gfCNCPoint2[4835] = {X 398.4217, Y 43.2753, Z -2.1667, A 0.000, B 0.000, C 0.000 }
gfCNCPoint2[4836] = {X 398.7237, Y 42.4397, Z -2.1667, A 0.000, B 0.000, C 0.000 }
gfCNCPoint2[4837] = {X 399.2028, Y 41.6913, Z -2.1667, A 0.000, B 0.000, C 0.000 }
gfCNCPoint2[4838] = {X 399.8352, Y 41.0672, Z -2.1667, A 0.000, B 0.000, C 0.000 }
gfCNCPoint2[4839] = {X 399.8352, Y 31.6238, Z -2.1667, A 0.000, B 0.000, C 0.000 }
gfCNCPoint2[4840] = {X 399.8383, Y 31.5919, Z -2.1667, A 0.000, B 0.000, C 0.000 }
gfCNCPoint2[4841] = {X 393.5981, Y 20.7408, Z -2.1667, A 0.000, B 0.000, C 0.000 }
gfCNCPoint2[4842] = {X 392.7769, Y 19.3501, Z -2.1667, A 0.000, B 0.000, C 0.000 }
gfCNCPoint2[4843] = {X 391.9239, Y 17.9787, Z -2.1667, A 0.000, B 0.000, C 0.000 }
gfCNCPoint2[4844] = {X 391.4254, Y 17.2996, Z -2.1667, A 0.000, B 0.000, C 0.000 }
gfCNCPoint2[4845] = {X 390.8426, Y 16.6913, Z -2.1667, A 0.000, B 0.000, C 0.000 }
gfCNCPoint2[4846] = {X 390.0091, Y 16.2361, Z -2.1667, A 0.000, B 0.000, C 0.000 }
gfCNCPoint2[4847] = {X 389.3064, Y 15.5972, Z -2.1667, A 0.000, B 0.000, C 0.000 }
gfCNCPoint2[4848] = {X 388.7742, Y 14.8107, Z -2.1667, A 0.000, B 0.000, C 0.000 }
gfCNCPoint2[4849] = {X 388.4423, Y 13.9209, Z -2.1667, A 0.000, B 0.000, C 0.000 }
gfCNCPoint2[4850] = {X 388.3296, Y 12.9779, Z -2.1667, A 0.000, B 0.000, C 0.000 }
gfCNCPoint2[4851] = {X 388.3296, Y 12.1868, Z -2.1667, A 0.000, B 0.000, C 0.000 }
gfCNCPoint2[4852] = {X 388.4299, Y 11.2967, Z -2.1667, A 0.000, B 0.000, C 0.000 }
gfCNCPoint2[4853] = {X 388.7258, Y 10.4513, Z -2.1667, A 0.000, B 0.000, C 0.000 }
gfCNCPoint2[4854] = {X 389.2023, Y 9.6929, Z -2.1667, A 0.000, B 0.000, C 0.000 }
gfCNCPoint2[4855] = {X 389.8357, Y 9.0595, Z -2.1667, A 0.000, B 0.000, C 0.000 }
gfCNCPoint2[4856] = {X 390.5941, Y 8.5829, Z -2.1667, A 0.000, B 0.000, C 0.000 }
gfCNCPoint2[4857] = {X 391.4395, Y 8.2871, Z -2.1667, A 0.000, B 0.000, C 0.000 }
gfCNCPoint2[4858] = {X 392.3296, Y 8.1868, Z -2.1667, A 0.000, B 0.000, C 0.000 }
gfCNCPoint2[4859] = {X 399.1118, Y 8.1868, Z -2.1667, A 0.000, B 0.000, C 0.000 }
gfCNCPoint2[4860] = {X 400.0018, Y 8.2871, Z -2.1667, A 0.000, B 0.000, C 0.000 }
gfCNCPoint2[4861] = {X 400.8473, Y 8.5829, Z -2.1667, A 0.000, B 0.000, C 0.000 }
gfCNCPoint2[4862] = {X 401.6057, Y 9.0595, Z -2.1667, A 0.000, B 0.000, C 0.000 }
gfCNCPoint2[4863] = {X 402.2391, Y 9.6929, Z -2.1667, A 0.000, B 0.000, C 0.000 }
gfCNCPoint2[4864] = {X 402.7156, Y 10.4513, Z -2.1667, A 0.000, B 0.000, C 0.000 }
gfCNCPoint2[4865] = {X 403.0115, Y 11.2967, Z -2.1667, A 0.000, B 0.000, C 0.000 }
gfCNCPoint2[4866] = {X 403.1118, Y 12.1868, Z -2.1667, A 0.000, B 0.000, C 0.000 }
gfCNCPoint2[4867] = {X 403.1115, Y 13.0192, Z -2.1667, A 0.000, B 0.000, C 0.000 }
gfCNCPoint2[4868] = {X 402.9933, Y 13.9442, Z -2.1667, A 0.000, B 0.000, C 0.000 }
gfCNCPoint2[4869] = {X 402.6641, Y 14.8167, Z -2.1667, A 0.000, B 0.000, C 0.000 }
gfCNCPoint2[4870] = {X 405.2576, Y 19.3199, Z -2.1667, A 0.000, B 0.000, C 0.000 }
gfCNCPoint2[4871] = {X 405.3717, Y 19.4085, Z -2.1667, A 0.000, B 0.000, C 0.000 }
gfCNCPoint2[4872] = {X 408.1956, Y 14.8342, Z -2.1667, A 0.000, B 0.000, C 0.000 }
gfCNCPoint2[4873] = {X 408.2428, Y 14.7847, Z -2.1667, A 0.000, B 0.000, C 0.000 }
gfCNCPoint2[4874] = {X 408.1939, Y 14.6846, Z -2.1667, A 0.000, B 0.000, C 0.000 }
gfCNCPoint2[4875] = {X 408.1478, Y 14.5832, Z -2.1667, A 0.000, B 0.000, C 0.000 }
gfCNCPoint2[4876] = {X 407.8965, Y 13.7980, Z -2.1667, A 0.000, B 0.000, C 0.000 }
gfCNCPoint2[4877] = {X 407.8115, Y 12.9779, Z -2.1667, A 0.000, B 0.000, C 0.000 }
gfCNCPoint2[4878] = {X 407.8115, Y 12.1868, Z -2.1667, A 0.000, B 0.000, C 0.000 }
gfCNCPoint2[4879] = {X 407.9118, Y 11.2967, Z -2.1667, A 0.000, B 0.000, C 0.000 }
gfCNCPoint2[4880] = {X 408.2077, Y 10.4513, Z -2.1667, A 0.000, B 0.000, C 0.000 }
gfCNCPoint2[4881] = {X 408.6842, Y 9.6929, Z -2.1667, A 0.000, B 0.000, C 0.000 }
gfCNCPoint2[4882] = {X 409.3176, Y 9.0595, Z -2.1667, A 0.000, B 0.000, C 0.000 }
gfCNCPoint2[4883] = {X 410.0760, Y 8.5829, Z -2.1667, A 0.000, B 0.000, C 0.000 }
gfCNCPoint2[4884] = {X 410.9215, Y 8.2871, Z -2.1667, A 0.000, B 0.000, C 0.000 }
gfCNCPoint2[4885] = {X 411.8115, Y 8.1868, Z -2.1667, A 0.000, B 0.000, C 0.000 }
gfCNCPoint2[4886] = {X 419.3245, Y 8.1868, Z -2.1667, A 0.000, B 0.000, C 0.000 }
gfCNCPoint2[4887] = {X 420.2145, Y 8.2871, Z -2.1667, A 0.000, B 0.000, C 0.000 }
gfCNCPoint2[4888] = {X 421.0600, Y 8.5829, Z -2.1667, A 0.000, B 0.000, C 0.000 }
gfCNCPoint2[4889] = {X 421.8184, Y 9.0595, Z -2.1667, A 0.000, B 0.000, C 0.000 }
gfCNCPoint2[4890] = {X 422.4518, Y 9.6929, Z -2.1667, A 0.000, B 0.000, C 0.000 }
gfCNCPoint2[4891] = {X 422.9283, Y 10.4513, Z -2.1667, A 0.000, B 0.000, C 0.000 }
gfCNCPoint2[4892] = {X 423.2242, Y 11.2967, Z -2.1667, A 0.000, B 0.000, C 0.000 }
gfCNCPoint2[4893] = {X 423.3245, Y 12.1868, Z -2.1667, A 0.000, B 0.000, C 0.000 }
gfCNCPoint2[4894] = {X 423.3245, Y 12.9779, Z -2.1667, A 0.000, B 0.000, C 0.000 }
gfCNCPoint2[4895] = {X 423.1973, Y 13.9553, Z -2.1667, A 0.000, B 0.000, C 0.000 }
gfCNCPoint2[4896] = {X 422.8388, Y 14.8734, Z -2.1667, A 0.000, B 0.000, C 0.000 }
gfCNCPoint2[4897] = {X 422.2699, Y 15.6782, Z -2.1667, A 0.000, B 0.000, C 0.000 }
gfCNCPoint2[4898] = {X 421.5242, Y 16.3226, Z -2.1667, A 0.000, B 0.000, C 0.000 }
gfCNCPoint2[4899] = {X 420.6453, Y 16.7687, Z -2.1667, A 0.000, B 0.000, C 0.000 }
gfCNCPoint2[4900] = {X 419.8864, Y 17.7815, Z -2.1667, A 0.000, B 0.000, C 0.000 }
gfCNCPoint2[4901] = {X 419.2015, Y 18.8457, Z -2.1667, A 0.000, B 0.000, C 0.000 }
gfCNCPoint2[4902] = {X 417.7223, Y 21.2414, Z -2.1667, A 0.000, B 0.000, C 0.000 }
gfCNCPoint2[4903] = {X 415.8783, Y 24.2025, Z -2.1667, A 0.000, B 0.000, C 0.000 }
gfCNCPoint2[4904] = {X 419.3417, Y 26.3592, Z -2.1667, A 0.000, B 0.000, C 0.000 }
gfCNCPoint2[4905] = {X 419.3417, Y 26.3592, Z 0.8333, A 0.000, B 0.000, C 0.000 }
gfCNCPoint2[4906] = {X 419.3417, Y 26.3592, Z 11.0000, A 0.000, B 0.000, C 0.000 }
gfCNCPoint2[4907] = {X 352.3279, Y -3.5331, Z 11.0000, A 0.000, B 0.000, C 0.000 }
gfCNCPoint2[4908] = {X 352.3279, Y -3.5331, Z 0.8333, A 0.000, B 0.000, C 0.000 }
gfCNCPoint2[4909] = {X 352.3279, Y -3.5331, Z -2.1667, A 0.000, B 0.000, C 0.000 }
gfCNCPoint2[4910] = {X 351.5857, Y 0.4789, Z -2.1667, A 0.000, B 0.000, C 0.000 }
gfCNCPoint2[4911] = {X 351.8688, Y 0.5312, Z -2.1667, A 0.000, B 0.000, C 0.000 }
gfCNCPoint2[4912] = {X 353.8034, Y 1.0172, Z -2.1667, A 0.000, B 0.000, C 0.000 }
gfCNCPoint2[4913] = {X 355.6832, Y 1.6844, Z -2.1667, A 0.000, B 0.000, C 0.000 }
gfCNCPoint2[4914] = {X 357.4913, Y 2.5267, Z -2.1667, A 0.000, B 0.000, C 0.000 }
gfCNCPoint2[4915] = {X 359.2115, Y 3.5365, Z -2.1667, A 0.000, B 0.000, C 0.000 }
gfCNCPoint2[4916] = {X 360.8283, Y 4.7047, Z -2.1667, A 0.000, B 0.000, C 0.000 }
gfCNCPoint2[4917] = {X 362.3270, Y 6.0209, Z -2.1667, A 0.000, B 0.000, C 0.000 }
gfCNCPoint2[4918] = {X 363.6944, Y 7.4732, Z -2.1667, A 0.000, B 0.000, C 0.000 }
gfCNCPoint2[4919] = {X 365.1629, Y 9.3684, Z -2.1667, A 0.000, B 0.000, C 0.000 }
gfCNCPoint2[4920] = {X 366.4410, Y 11.3969, Z -2.1667, A 0.000, B 0.000, C 0.000 }
gfCNCPoint2[4921] = {X 367.5165, Y 13.5398, Z -2.1667, A 0.000, B 0.000, C 0.000 }
gfCNCPoint2[4922] = {X 368.3793, Y 15.7767, Z -2.1667, A 0.000, B 0.000, C 0.000 }
gfCNCPoint2[4923] = {X 369.0214, Y 18.0867, Z -2.1667, A 0.000, B 0.000, C 0.000 }
gfCNCPoint2[4924] = {X 369.5013, Y 20.7195, Z -2.1667, A 0.000, B 0.000, C 0.000 }
gfCNCPoint2[4925] = {X 369.7569, Y 23.3834, Z -2.1667, A 0.000, B 0.000, C 0.000 }
gfCNCPoint2[4926] = {X 369.7864, Y 26.0594, Z -2.1667, A 0.000, B 0.000, C 0.000 }
gfCNCPoint2[4927] = {X 369.5897, Y 28.7284, Z -2.1667, A 0.000, B 0.000, C 0.000 }
gfCNCPoint2[4928] = {X 369.1680, Y 31.3711, Z -2.1667, A 0.000, B 0.000, C 0.000 }
gfCNCPoint2[4929] = {X 368.6442, Y 33.4757, Z -2.1667, A 0.000, B 0.000, C 0.000 }
gfCNCPoint2[4930] = {X 367.9363, Y 35.5257, Z -2.1667, A 0.000, B 0.000, C 0.000 }
gfCNCPoint2[4931] = {X 367.0501, Y 37.5052, Z -2.1667, A 0.000, B 0.000, C 0.000 }
gfCNCPoint2[4932] = {X 365.9924, Y 39.3986, Z -2.1667, A 0.000, B 0.000, C 0.000 }
gfCNCPoint2[4933] = {X 364.7715, Y 41.1911, Z -2.1667, A 0.000, B 0.000, C 0.000 }
gfCNCPoint2[4934] = {X 363.5445, Y 42.7031, Z -2.1667, A 0.000, B 0.000, C 0.000 }
gfCNCPoint2[4935] = {X 362.1896, Y 44.1017, Z -2.1667, A 0.000, B 0.000, C 0.000 }
gfCNCPoint2[4936] = {X 360.7172, Y 45.3761, Z -2.1667, A 0.000, B 0.000, C 0.000 }
gfCNCPoint2[4937] = {X 359.1388, Y 46.5165, Z -2.1667, A 0.000, B 0.000, C 0.000 }
gfCNCPoint2[4938] = {X 357.4664, Y 47.5140, Z -2.1667, A 0.000, B 0.000, C 0.000 }
gfCNCPoint2[4939] = {X 355.5058, Y 48.4044, Z -2.1667, A 0.000, B 0.000, C 0.000 }
gfCNCPoint2[4940] = {X 353.4695, Y 49.1044, Z -2.1667, A 0.000, B 0.000, C 0.000 }
gfCNCPoint2[4941] = {X 351.3759, Y 49.6077, Z -2.1667, A 0.000, B 0.000, C 0.000 }
gfCNCPoint2[4942] = {X 349.2439, Y 49.9098, Z -2.1667, A 0.000, B 0.000, C 0.000 }
gfCNCPoint2[4943] = {X 347.0929, Y 50.0079, Z -2.1667, A 0.000, B 0.000, C 0.000 }
gfCNCPoint2[4944] = {X 345.0263, Y 49.9731, Z -2.1667, A 0.000, B 0.000, C 0.000 }
gfCNCPoint2[4945] = {X 342.9706, Y 49.7591, Z -2.1667, A 0.000, B 0.000, C 0.000 }
gfCNCPoint2[4946] = {X 340.9411, Y 49.3676, Z -2.1667, A 0.000, B 0.000, C 0.000 }
gfCNCPoint2[4947] = {X 338.9533, Y 48.8016, Z -2.1667, A 0.000, B 0.000, C 0.000 }
gfCNCPoint2[4948] = {X 337.0220, Y 48.0653, Z -2.1667, A 0.000, B 0.000, C 0.000 }
gfCNCPoint2[4949] = {X 335.1619, Y 47.1643, Z -2.1667, A 0.000, B 0.000, C 0.000 }
gfCNCPoint2[4950] = {X 333.5788, Y 46.1857, Z -2.1667, A 0.000, B 0.000, C 0.000 }
gfCNCPoint2[4951] = {X 332.0761, Y 45.0877, Z -2.1667, A 0.000, B 0.000, C 0.000 }
gfCNCPoint2[4952] = {X 330.6627, Y 43.8770, Z -2.1667, A 0.000, B 0.000, C 0.000 }
gfCNCPoint2[4953] = {X 329.7215, Y 43.8765, Z -2.1667, A 0.000, B 0.000, C 0.000 }
gfCNCPoint2[4954] = {X 328.8028, Y 43.6722, Z -2.1667, A 0.000, B 0.000, C 0.000 }
gfCNCPoint2[4955] = {X 327.9502, Y 43.2738, Z -2.1667, A 0.000, B 0.000, C 0.000 }
gfCNCPoint2[4956] = {X 327.2040, Y 42.7002, Z -2.1667, A 0.000, B 0.000, C 0.000 }
gfCNCPoint2[4957] = {X 326.5808, Y 42.0925, Z -2.1667, A 0.000, B 0.000, C 0.000 }
gfCNCPoint2[4958] = {X 325.9523, Y 41.3190, Z -2.1667, A 0.000, B 0.000, C 0.000 }
gfCNCPoint2[4959] = {X 325.5179, Y 40.4220, Z -2.1667, A 0.000, B 0.000, C 0.000 }
gfCNCPoint2[4960] = {X 325.3006, Y 39.4493, Z -2.1667, A 0.000, B 0.000, C 0.000 }
gfCNCPoint2[4961] = {X 325.3120, Y 38.4527, Z -2.1667, A 0.000, B 0.000, C 0.000 }
gfCNCPoint2[4962] = {X 325.5514, Y 37.4852, Z -2.1667, A 0.000, B 0.000, C 0.000 }
gfCNCPoint2[4963] = {X 326.0062, Y 36.5984, Z -2.1667, A 0.000, B 0.000, C 0.000 }
gfCNCPoint2[4964] = {X 330.2648, Y 30.2313, Z -2.1667, A 0.000, B 0.000, C 0.000 }
gfCNCPoint2[4965] = {X 330.8696, Y 29.5246, Z -2.1667, A 0.000, B 0.000, C 0.000 }
gfCNCPoint2[4966] = {X 331.6116, Y 28.9637, Z -2.1667, A 0.000, B 0.000, C 0.000 }
gfCNCPoint2[4967] = {X 332.4564, Y 28.5747, Z -2.1667, A 0.000, B 0.000, C 0.000 }
gfCNCPoint2[4968] = {X 333.3649, Y 28.3755, Z -2.1667, A 0.000, B 0.000, C 0.000 }
gfCNCPoint2[4969] = {X 334.2951, Y 28.3754, Z -2.1667, A 0.000, B 0.000, C 0.000 }
gfCNCPoint2[4970] = {X 335.2036, Y 28.5744, Z -2.1667, A 0.000, B 0.000, C 0.000 }
gfCNCPoint2[4971] = {X 336.0486, Y 28.9633, Z -2.1667, A 0.000, B 0.000, C 0.000 }
gfCNCPoint2[4972] = {X 336.7907, Y 29.5240, Z -2.1667, A 0.000, B 0.000, C 0.000 }
gfCNCPoint2[4973] = {X 337.4284, Y 30.1382, Z -2.1667, A 0.000, B 0.000, C 0.000 }
gfCNCPoint2[4974] = {X 337.9530, Y 30.7613, Z -2.1667, A 0.000, B 0.000, C 0.000 }
gfCNCPoint2[4975] = {X 338.3513, Y 31.4717, Z -2.1667, A 0.000, B 0.000, C 0.000 }
gfCNCPoint2[4976] = {X 338.6092, Y 32.2443, Z -2.1667, A 0.000, B 0.000, C 0.000 }
gfCNCPoint2[4977] = {X 338.7175, Y 33.0516, Z -2.1667, A 0.000, B 0.000, C 0.000 }
gfCNCPoint2[4978] = {X 338.6724, Y 33.8648, Z -2.1667, A 0.000, B 0.000, C 0.000 }
gfCNCPoint2[4979] = {X 339.4354, Y 34.5563, Z -2.1667, A 0.000, B 0.000, C 0.000 }
gfCNCPoint2[4980] = {X 340.2328, Y 35.2080, Z -2.1667, A 0.000, B 0.000, C 0.000 }
gfCNCPoint2[4981] = {X 341.5301, Y 36.0603, Z -2.1667, A 0.000, B 0.000, C 0.000 }
gfCNCPoint2[4982] = {X 342.9378, Y 36.7142, Z -2.1667, A 0.000, B 0.000, C 0.000 }
gfCNCPoint2[4983] = {X 344.4258, Y 37.1559, Z -2.1667, A 0.000, B 0.000, C 0.000 }
gfCNCPoint2[4984] = {X 345.9624, Y 37.3758, Z -2.1667, A 0.000, B 0.000, C 0.000 }
gfCNCPoint2[4985] = {X 347.5146, Y 37.3693, Z -2.1667, A 0.000, B 0.000, C 0.000 }
gfCNCPoint2[4986] = {X 348.9586, Y 37.1756, Z -2.1667, A 0.000, B 0.000, C 0.000 }
gfCNCPoint2[4987] = {X 350.3516, Y 36.7489, Z -2.1667, A 0.000, B 0.000, C 0.000 }
gfCNCPoint2[4988] = {X 351.6563, Y 36.1004, Z -2.1667, A 0.000, B 0.000, C 0.000 }
gfCNCPoint2[4989] = {X 352.8377, Y 35.2478, Z -2.1667, A 0.000, B 0.000, C 0.000 }
gfCNCPoint2[4990] = {X 353.9885, Y 34.1272, Z -2.1667, A 0.000, B 0.000, C 0.000 }
gfCNCPoint2[4991] = {X 354.9846, Y 32.8671, Z -2.1667, A 0.000, B 0.000, C 0.000 }
gfCNCPoint2[4992] = {X 355.8091, Y 31.4886, Z -2.1667, A 0.000, B 0.000, C 0.000 }
gfCNCPoint2[4993] = {X 356.4482, Y 30.0150, Z -2.1667, A 0.000, B 0.000, C 0.000 }
gfCNCPoint2[4994] = {X 356.8912, Y 28.4710, Z -2.1667, A 0.000, B 0.000, C 0.000 }
gfCNCPoint2[4995] = {X 357.1644, Y 26.7828, Z -2.1667, A 0.000, B 0.000, C 0.000 }
gfCNCPoint2[4996] = {X 357.2757, Y 25.0763, Z -2.1667, A 0.000, B 0.000, C 0.000 }
gfCNCPoint2[4997] = {X 357.2241, Y 23.3669, Z -2.1667, A 0.000, B 0.000, C 0.000 }
gfCNCPoint2[4998] = {X 357.0099, Y 21.6701, Z -2.1667, A 0.000, B 0.000, C 0.000 }
gfCNCPoint2[4999] = {X 356.6736, Y 20.2206, Z -2.1667, A 0.000, B 0.000, C 0.000 }
gfCNCPoint2[5000] = {X 356.1606, Y 18.8238, Z -2.1667, A 0.000, B 0.000, C 0.000 }
gfCNCPoint2[5001] = {X 355.4786, Y 17.5012, Z -2.1667, A 0.000, B 0.000, C 0.000 }
gfCNCPoint2[5002] = {X 354.6382, Y 16.2732, Z -2.1667, A 0.000, B 0.000, C 0.000 }
gfCNCPoint2[5003] = {X 353.7522, Y 15.2850, Z -2.1667, A 0.000, B 0.000, C 0.000 }
gfCNCPoint2[5004] = {X 352.7339, Y 14.4340, Z -2.1667, A 0.000, B 0.000, C 0.000 }
gfCNCPoint2[5005] = {X 351.6041, Y 13.7377, Z -2.1667, A 0.000, B 0.000, C 0.000 }
gfCNCPoint2[5006] = {X 350.3862, Y 13.2104, Z -2.1667, A 0.000, B 0.000, C 0.000 }
gfCNCPoint2[5007] = {X 349.1053, Y 12.8630, Z -2.1667, A 0.000, B 0.000, C 0.000 }
gfCNCPoint2[5008] = {X 347.3447, Y 12.6441, Z -2.1667, A 0.000, B 0.000, C 0.000 }
gfCNCPoint2[5009] = {X 345.5707, Y 12.6601, Z -2.1667, A 0.000, B 0.000, C 0.000 }
gfCNCPoint2[5010] = {X 343.8144, Y 12.9106, Z -2.1667, A 0.000, B 0.000, C 0.000 }
gfCNCPoint2[5011] = {X 342.1066, Y 13.3911, Z -2.1667, A 0.000, B 0.000, C 0.000 }
gfCNCPoint2[5012] = {X 340.4774, Y 14.0933, Z -2.1667, A 0.000, B 0.000, C 0.000 }
gfCNCPoint2[5013] = {X 338.9554, Y 15.0048, Z -2.1667, A 0.000, B 0.000, C 0.000 }
gfCNCPoint2[5014] = {X 338.9168, Y 15.8495, Z -2.1667, A 0.000, B 0.000, C 0.000 }
gfCNCPoint2[5015] = {X 338.7144, Y 16.6705, Z -2.1667, A 0.000, B 0.000, C 0.000 }
gfCNCPoint2[5016] = {X 338.3559, Y 17.4363, Z -2.1667, A 0.000, B 0.000, C 0.000 }
gfCNCPoint2[5017] = {X 337.8551, Y 18.1177, Z -2.1667, A 0.000, B 0.000, C 0.000 }
gfCNCPoint2[5018] = {X 337.2313, Y 18.6884, Z -2.1667, A 0.000, B 0.000, C 0.000 }
gfCNCPoint2[5019] = {X 336.5140, Y 19.2162, Z -2.1667, A 0.000, B 0.000, C 0.000 }
gfCNCPoint2[5020] = {X 335.6982, Y 19.6754, Z -2.1667, A 0.000, B 0.000, C 0.000 }
gfCNCPoint2[5021] = {X 334.8027, Y 19.9480, Z -2.1667, A 0.000, B 0.000, C 0.000 }
gfCNCPoint2[5022] = {X 333.8694, Y 20.0213, Z -2.1667, A 0.000, B 0.000, C 0.000 }
gfCNCPoint2[5023] = {X 332.9422, Y 19.8919, Z -2.1667, A 0.000, B 0.000, C 0.000 }
gfCNCPoint2[5024] = {X 332.0647, Y 19.5657, Z -2.1667, A 0.000, B 0.000, C 0.000 }
gfCNCPoint2[5025] = {X 331.2781, Y 19.0581, Z -2.1667, A 0.000, B 0.000, C 0.000 }
gfCNCPoint2[5026] = {X 330.6193, Y 18.3931, Z -2.1667, A 0.000, B 0.000, C 0.000 }
gfCNCPoint2[5027] = {X 330.1192, Y 17.6017, Z -2.1667, A 0.000, B 0.000, C 0.000 }
gfCNCPoint2[5028] = {X 326.5942, Y 10.3502, Z -2.1667, A 0.000, B 0.000, C 0.000 }
gfCNCPoint2[5029] = {X 326.2930, Y 9.5271, Z -2.1667, A 0.000, B 0.000, C 0.000 }
gfCNCPoint2[5030] = {X 326.1640, Y 8.6602, Z -2.1667, A 0.000, B 0.000, C 0.000 }
gfCNCPoint2[5031] = {X 326.2128, Y 7.7851, Z -2.1667, A 0.000, B 0.000, C 0.000 }
gfCNCPoint2[5032] = {X 326.4371, Y 6.9378, Z -2.1667, A 0.000, B 0.000, C 0.000 }
gfCNCPoint2[5033] = {X 326.8279, Y 6.1532, Z -2.1667, A 0.000, B 0.000, C 0.000 }
gfCNCPoint2[5034] = {X 327.3690, Y 5.4637, Z -2.1667, A 0.000, B 0.000, C 0.000 }
gfCNCPoint2[5035] = {X 328.0381, Y 4.8976, Z -2.1667, A 0.000, B 0.000, C 0.000 }
gfCNCPoint2[5036] = {X 328.7084, Y 4.4385, Z -2.1667, A 0.000, B 0.000, C 0.000 }
gfCNCPoint2[5037] = {X 329.5890, Y 3.9826, Z -2.1667, A 0.000, B 0.000, C 0.000 }
gfCNCPoint2[5038] = {X 330.5503, Y 3.7395, Z -2.1667, A 0.000, B 0.000, C 0.000 }
gfCNCPoint2[5039] = {X 331.5417, Y 3.7221, Z -2.1667, A 0.000, B 0.000, C 0.000 }
gfCNCPoint2[5040] = {X 332.5111, Y 3.9311, Z -2.1667, A 0.000, B 0.000, C 0.000 }
gfCNCPoint2[5041] = {X 333.9977, Y 3.1015, Z -2.1667, A 0.000, B 0.000, C 0.000 }
gfCNCPoint2[5042] = {X 335.5315, Y 2.3626, Z -2.1667, A 0.000, B 0.000, C 0.000 }
gfCNCPoint2[5043] = {X 337.6677, Y 1.4960, Z -2.1667, A 0.000, B 0.000, C 0.000 }
gfCNCPoint2[5044] = {X 339.8716, Y 0.8200, Z -2.1667, A 0.000, B 0.000, C 0.000 }
gfCNCPoint2[5045] = {X 342.1263, Y 0.3396, Z -2.1667, A 0.000, B 0.000, C 0.000 }
gfCNCPoint2[5046] = {X 344.4143, Y 0.0587, Z -2.1667, A 0.000, B 0.000, C 0.000 }
gfCNCPoint2[5047] = {X 346.7182, Y -0.0206, Z -2.1667, A 0.000, B 0.000, C 0.000 }
gfCNCPoint2[5048] = {X 349.0202, Y 0.1023, Z -2.1667, A 0.000, B 0.000, C 0.000 }
gfCNCPoint2[5049] = {X 351.3025, Y 0.4265, Z -2.1667, A 0.000, B 0.000, C 0.000 }
gfCNCPoint2[5050] = {X 351.5857, Y 0.4789, Z -2.1667, A 0.000, B 0.000, C 0.000 }
gfCNCPoint2[5051] = {X 352.3133, Y -3.4544, Z -2.1667, A 0.000, B 0.000, C 0.000 }
gfCNCPoint2[5052] = {X 351.5711, Y 0.5575, Z -2.1667, A 0.000, B 0.000, C 0.000 }
gfCNCPoint2[5053] = {X 351.8536, Y 0.6098, Z -2.1667, A 0.000, B 0.000, C 0.000 }
gfCNCPoint2[5054] = {X 353.7807, Y 1.0940, Z -2.1667, A 0.000, B 0.000, C 0.000 }
gfCNCPoint2[5055] = {X 355.6533, Y 1.7586, Z -2.1667, A 0.000, B 0.000, C 0.000 }
gfCNCPoint2[5056] = {X 357.4544, Y 2.5977, Z -2.1667, A 0.000, B 0.000, C 0.000 }
gfCNCPoint2[5057] = {X 359.1680, Y 3.6036, Z -2.1667, A 0.000, B 0.000, C 0.000 }
gfCNCPoint2[5058] = {X 360.7785, Y 4.7674, Z -2.1667, A 0.000, B 0.000, C 0.000 }
gfCNCPoint2[5059] = {X 362.2715, Y 6.0785, Z -2.1667, A 0.000, B 0.000, C 0.000 }
gfCNCPoint2[5060] = {X 363.6336, Y 7.5252, Z -2.1667, A 0.000, B 0.000, C 0.000 }
gfCNCPoint2[5061] = {X 365.0974, Y 9.4143, Z -2.1667, A 0.000, B 0.000, C 0.000 }
gfCNCPoint2[5062] = {X 366.3713, Y 11.4363, Z -2.1667, A 0.000, B 0.000, C 0.000 }
gfCNCPoint2[5063] = {X 367.4433, Y 13.5721, Z -2.1667, A 0.000, B 0.000, C 0.000 }
gfCNCPoint2[5064] = {X 368.3034, Y 15.8018, Z -2.1667, A 0.000, B 0.000, C 0.000 }
gfCNCPoint2[5065] = {X 368.9434, Y 18.1043, Z -2.1667, A 0.000, B 0.000, C 0.000 }
gfCNCPoint2[5066] = {X 369.4221, Y 20.7305, Z -2.1667, A 0.000, B 0.000, C 0.000 }
gfCNCPoint2[5067] = {X 369.6770, Y 23.3877, Z -2.1667, A 0.000, B 0.000, C 0.000 }
gfCNCPoint2[5068] = {X 369.7065, Y 26.0569, Z -2.1667, A 0.000, B 0.000, C 0.000 }
gfCNCPoint2[5069] = {X 369.5102, Y 28.7191, Z -2.1667, A 0.000, B 0.000, C 0.000 }
gfCNCPoint2[5070] = {X 369.0896, Y 31.3552, Z -2.1667, A 0.000, B 0.000, C 0.000 }
gfCNCPoint2[5071] = {X 368.5675, Y 33.4529, Z -2.1667, A 0.000, B 0.000, C 0.000 }
gfCNCPoint2[5072] = {X 367.8619, Y 35.4963, Z -2.1667, A 0.000, B 0.000, C 0.000 }
gfCNCPoint2[5073] = {X 366.9786, Y 37.4694, Z -2.1667, A 0.000, B 0.000, C 0.000 }
gfCNCPoint2[5074] = {X 365.9243, Y 39.3566, Z -2.1667, A 0.000, B 0.000, C 0.000 }
gfCNCPoint2[5075] = {X 364.7073, Y 41.1433, Z -2.1667, A 0.000, B 0.000, C 0.000 }
gfCNCPoint2[5076] = {X 363.4848, Y 42.6498, Z -2.1667, A 0.000, B 0.000, C 0.000 }
gfCNCPoint2[5077] = {X 362.1349, Y 44.0433, Z -2.1667, A 0.000, B 0.000, C 0.000 }
gfCNCPoint2[5078] = {X 360.6680, Y 45.3131, Z -2.1667, A 0.000, B 0.000, C 0.000 }
gfCNCPoint2[5079] = {X 359.0954, Y 46.4493, Z -2.1667, A 0.000, B 0.000, C 0.000 }
gfCNCPoint2[5080] = {X 357.4292, Y 47.4432, Z -2.1667, A 0.000, B 0.000, C 0.000 }
gfCNCPoint2[5081] = {X 355.4754, Y 48.3304, Z -2.1667, A 0.000, B 0.000, C 0.000 }
gfCNCPoint2[5082] = {X 353.4462, Y 49.0279, Z -2.1667, A 0.000, B 0.000, C 0.000 }
gfCNCPoint2[5083] = {X 351.3599, Y 49.5293, Z -2.1667, A 0.000, B 0.000, C 0.000 }
gfCNCPoint2[5084] = {X 349.2354, Y 49.8303, Z -2.1667, A 0.000, B 0.000, C 0.000 }
gfCNCPoint2[5085] = {X 347.0919, Y 49.9279, Z -2.1667, A 0.000, B 0.000, C 0.000 }
gfCNCPoint2[5086] = {X 345.0322, Y 49.8933, Z -2.1667, A 0.000, B 0.000, C 0.000 }
gfCNCPoint2[5087] = {X 342.9833, Y 49.6801, Z -2.1667, A 0.000, B 0.000, C 0.000 }
gfCNCPoint2[5088] = {X 340.9606, Y 49.2900, Z -2.1667, A 0.000, B 0.000, C 0.000 }
gfCNCPoint2[5089] = {X 338.9794, Y 48.7260, Z -2.1667, A 0.000, B 0.000, C 0.000 }
gfCNCPoint2[5090] = {X 337.0546, Y 47.9922, Z -2.1667, A 0.000, B 0.000, C 0.000 }
gfCNCPoint2[5091] = {X 335.2006, Y 47.0943, Z -2.1667, A 0.000, B 0.000, C 0.000 }
gfCNCPoint2[5092] = {X 333.6129, Y 46.1122, Z -2.1667, A 0.000, B 0.000, C 0.000 }
gfCNCPoint2[5093] = {X 332.1064, Y 45.0097, Z -2.1667, A 0.000, B 0.000, C 0.000 }
gfCNCPoint2[5094] = {X 330.6901, Y 43.7933, Z -2.1667, A 0.000, B 0.000, C 0.000 }
gfCNCPoint2[5095] = {X 329.7574, Y 43.7998, Z -2.1667, A 0.000, B 0.000, C 0.000 }
gfCNCPoint2[5096] = {X 328.8458, Y 43.6023, Z -2.1667, A 0.000, B 0.000, C 0.000 }
gfCNCPoint2[5097] = {X 327.9995, Y 43.2102, Z -2.1667, A 0.000, B 0.000, C 0.000 }
gfCNCPoint2[5098] = {X 327.2594, Y 42.6425, Z -2.1667, A 0.000, B 0.000, C 0.000 }
gfCNCPoint2[5099] = {X 326.6366, Y 42.0352, Z -2.1667, A 0.000, B 0.000, C 0.000 }
gfCNCPoint2[5100] = {X 326.0198, Y 41.2760, Z -2.1667, A 0.000, B 0.000, C 0.000 }
gfCNCPoint2[5101] = {X 325.5934, Y 40.3956, Z -2.1667, A 0.000, B 0.000, C 0.000 }
gfCNCPoint2[5102] = {X 325.3802, Y 39.4410, Z -2.1667, A 0.000, B 0.000, C 0.000 }
gfCNCPoint2[5103] = {X 325.3913, Y 38.4628, Z -2.1667, A 0.000, B 0.000, C 0.000 }
gfCNCPoint2[5104] = {X 325.6264, Y 37.5133, Z -2.1667, A 0.000, B 0.000, C 0.000 }
gfCNCPoint2[5105] = {X 326.0727, Y 36.6429, Z -2.1667, A 0.000, B 0.000, C 0.000 }
gfCNCPoint2[5106] = {X 330.3309, Y 30.2764, Z -2.1667, A 0.000, B 0.000, C 0.000 }
gfCNCPoint2[5107] = {X 330.9244, Y 29.5828, Z -2.1667, A 0.000, B 0.000, C 0.000 }
gfCNCPoint2[5108] = {X 331.6527, Y 29.0324, Z -2.1667, A 0.000, B 0.000, C 0.000 }
gfCNCPoint2[5109] = {X 332.4819, Y 28.6505, Z -2.1667, A 0.000, B 0.000, C 0.000 }
gfCNCPoint2[5110] = {X 333.3736, Y 28.4550, Z -2.1667, A 0.000, B 0.000, C 0.000 }
gfCNCPoint2[5111] = {X 334.2865, Y 28.4549, Z -2.1667, A 0.000, B 0.000, C 0.000 }
gfCNCPoint2[5112] = {X 335.1782, Y 28.6502, Z -2.1667, A 0.000, B 0.000, C 0.000 }
gfCNCPoint2[5113] = {X 336.0075, Y 29.0319, Z -2.1667, A 0.000, B 0.000, C 0.000 }
gfCNCPoint2[5114] = {X 336.7358, Y 29.5823, Z -2.1667, A 0.000, B 0.000, C 0.000 }
gfCNCPoint2[5115] = {X 337.3723, Y 30.1953, Z -2.1667, A 0.000, B 0.000, C 0.000 }
gfCNCPoint2[5116] = {X 337.8919, Y 30.8136, Z -2.1667, A 0.000, B 0.000, C 0.000 }
gfCNCPoint2[5117] = {X 338.2848, Y 31.5192, Z -2.1667, A 0.000, B 0.000, C 0.000 }
gfCNCPoint2[5118] = {X 338.5368, Y 32.2866, Z -2.1667, A 0.000, B 0.000, C 0.000 }
gfCNCPoint2[5119] = {X 338.6388, Y 33.0878, Z -2.1667, A 0.000, B 0.000, C 0.000 }
gfCNCPoint2[5120] = {X 338.5869, Y 33.8938, Z -2.1667, A 0.000, B 0.000, C 0.000 }
gfCNCPoint2[5121] = {X 339.3674, Y 34.6033, Z -2.1667, A 0.000, B 0.000, C 0.000 }
gfCNCPoint2[5122] = {X 340.1839, Y 35.2713, Z -2.1667, A 0.000, B 0.000, C 0.000 }
gfCNCPoint2[5123] = {X 341.4908, Y 36.1300, Z -2.1667, A 0.000, B 0.000, C 0.000 }
gfCNCPoint2[5124] = {X 342.9089, Y 36.7888, Z -2.1667, A 0.000, B 0.000, C 0.000 }
gfCNCPoint2[5125] = {X 344.4080, Y 37.2339, Z -2.1667, A 0.000, B 0.000, C 0.000 }
gfCNCPoint2[5126] = {X 345.9560, Y 37.4556, Z -2.1667, A 0.000, B 0.000, C 0.000 }
gfCNCPoint2[5127] = {X 347.5197, Y 37.4491, Z -2.1667, A 0.000, B 0.000, C 0.000 }
gfCNCPoint2[5128] = {X 348.6880, Y 37.3118, Z -2.1667, A 0.000, B 0.000, C 0.000 }
gfCNCPoint2[5129] = {X 349.8282, Y 37.0228, Z -2.1667, A 0.000, B 0.000, C 0.000 }
gfCNCPoint2[5130] = {X 350.9209, Y 36.5873, Z -2.1667, A 0.000, B 0.000, C 0.000 }
gfCNCPoint2[5131] = {X 351.9473, Y 36.0126, Z -2.1667, A 0.000, B 0.000, C 0.000 }
gfCNCPoint2[5132] = {X 352.8897, Y 35.3086, Z -2.1667, A 0.000, B 0.000, C 0.000 }
gfCNCPoint2[5133] = {X 354.0480, Y 34.1808, Z -2.1667, A 0.000, B 0.000, C 0.000 }
gfCNCPoint2[5134] = {X 355.0505, Y 32.9125, Z -2.1667, A 0.000, B 0.000, C 0.000 }
gfCNCPoint2[5135] = {X 355.8803, Y 31.5250, Z -2.1667, A 0.000, B 0.000, C 0.000 }
gfCNCPoint2[5136] = {X 356.5236, Y 30.0418, Z -2.1667, A 0.000, B 0.000, C 0.000 }
gfCNCPoint2[5137] = {X 356.9694, Y 28.4878, Z -2.1667, A 0.000, B 0.000, C 0.000 }
gfCNCPoint2[5138] = {X 357.2439, Y 26.7920, Z -2.1667, A 0.000, B 0.000, C 0.000 }
gfCNCPoint2[5139] = {X 357.3557, Y 25.0778, Z -2.1667, A 0.000, B 0.000, C 0.000 }
gfCNCPoint2[5140] = {X 357.3038, Y 23.3607, Z -2.1667, A 0.000, B 0.000, C 0.000 }
gfCNCPoint2[5141] = {X 357.0887, Y 21.6563, Z -2.1667, A 0.000, B 0.000, C 0.000 }
gfCNCPoint2[5142] = {X 356.7502, Y 20.1973, Z -2.1667, A 0.000, B 0.000, C 0.000 }
gfCNCPoint2[5143] = {X 356.2337, Y 18.7913, Z -2.1667, A 0.000, B 0.000, C 0.000 }
gfCNCPoint2[5144] = {X 355.5472, Y 17.4601, Z -2.1667, A 0.000, B 0.000, C 0.000 }
gfCNCPoint2[5145] = {X 354.7013, Y 16.2240, Z -2.1667, A 0.000, B 0.000, C 0.000 }
gfCNCPoint2[5146] = {X 353.8077, Y 15.2274, Z -2.1667, A 0.000, B 0.000, C 0.000 }
gfCNCPoint2[5147] = {X 352.7805, Y 14.3690, Z -2.1667, A 0.000, B 0.000, C 0.000 }
gfCNCPoint2[5148] = {X 351.6409, Y 13.6667, Z -2.1667, A 0.000, B 0.000, C 0.000 }
gfCNCPoint2[5149] = {X 350.4125, Y 13.1348, Z -2.1667, A 0.000, B 0.000, C 0.000 }
gfCNCPoint2[5150] = {X 349.1206, Y 12.7844, Z -2.1667, A 0.000, B 0.000, C 0.000 }
gfCNCPoint2[5151] = {X 347.3420, Y 12.5639, Z -2.1667, A 0.000, B 0.000, C 0.000 }
gfCNCPoint2[5152] = {X 345.5499, Y 12.5814, Z -2.1667, A 0.000, B 0.000, C 0.000 }
gfCNCPoint2[5153] = {X 343.7760, Y 12.8369, Z -2.1667, A 0.000, B 0.000, C 0.000 }
gfCNCPoint2[5154] = {X 342.0517, Y 13.3257, Z -2.1667, A 0.000, B 0.000, C 0.000 }
gfCNCPoint2[5155] = {X 340.4077, Y 14.0392, Z -2.1667, A 0.000, B 0.000, C 0.000 }
gfCNCPoint2[5156] = {X 338.8729, Y 14.9647, Z -2.1667, A 0.000, B 0.000, C 0.000 }
gfCNCPoint2[5157] = {X 338.8425, Y 15.8029, Z -2.1667, A 0.000, B 0.000, C 0.000 }
gfCNCPoint2[5158] = {X 338.6477, Y 16.6187, Z -2.1667, A 0.000, B 0.000, C 0.000 }
gfCNCPoint2[5159] = {X 338.2962, Y 17.3802, Z -2.1667, A 0.000, B 0.000, C 0.000 }
gfCNCPoint2[5160] = {X 337.8016, Y 18.0576, Z -2.1667, A 0.000, B 0.000, C 0.000 }
gfCNCPoint2[5161] = {X 337.1833, Y 18.6244, Z -2.1667, A 0.000, B 0.000, C 0.000 }
gfCNCPoint2[5162] = {X 336.4675, Y 19.1512, Z -2.1667, A 0.000, B 0.000, C 0.000 }
gfCNCPoint2[5163] = {X 335.6668, Y 19.6018, Z -2.1667, A 0.000, B 0.000, C 0.000 }
gfCNCPoint2[5164] = {X 334.7878, Y 19.8694, Z -2.1667, A 0.000, B 0.000, C 0.000 }
gfCNCPoint2[5165] = {X 333.8718, Y 19.9414, Z -2.1667, A 0.000, B 0.000, C 0.000 }
gfCNCPoint2[5166] = {X 332.9618, Y 19.8143, Z -2.1667, A 0.000, B 0.000, C 0.000 }
gfCNCPoint2[5167] = {X 332.1006, Y 19.4942, Z -2.1667, A 0.000, B 0.000, C 0.000 }
gfCNCPoint2[5168] = {X 331.3285, Y 18.9960, Z -2.1667, A 0.000, B 0.000, C 0.000 }
gfCNCPoint2[5169] = {X 330.6819, Y 18.3433, Z -2.1667, A 0.000, B 0.000, C 0.000 }
gfCNCPoint2[5170] = {X 330.1911, Y 17.5665, Z -2.1667, A 0.000, B 0.000, C 0.000 }
gfCNCPoint2[5171] = {X 326.6662, Y 10.3152, Z -2.1667, A 0.000, B 0.000, C 0.000 }
gfCNCPoint2[5172] = {X 326.3374, Y 9.3676, Z -2.1667, A 0.000, B 0.000, C 0.000 }
gfCNCPoint2[5173] = {X 326.2405, Y 8.3693, Z -2.1667, A 0.000, B 0.000, C 0.000 }
gfCNCPoint2[5174] = {X 326.3807, Y 7.3762, Z -2.1667, A 0.000, B 0.000, C 0.000 }
gfCNCPoint2[5175] = {X 326.7504, Y 6.4438, Z -2.1667, A 0.000, B 0.000, C 0.000 }
gfCNCPoint2[5176] = {X 327.3287, Y 5.6243, Z -2.1667, A 0.000, B 0.000, C 0.000 }
gfCNCPoint2[5177] = {X 328.0833, Y 4.9636, Z -2.1667, A 0.000, B 0.000, C 0.000 }
gfCNCPoint2[5178] = {X 328.7533, Y 4.5047, Z -2.1667, A 0.000, B 0.000, C 0.000 }
gfCNCPoint2[5179] = {X 329.6262, Y 4.0541, Z -2.1667, A 0.000, B 0.000, C 0.000 }
gfCNCPoint2[5180] = {X 330.5793, Y 3.8164, Z -2.1667, A 0.000, B 0.000, C 0.000 }
gfCNCPoint2[5181] = {X 331.5616, Y 3.8045, Z -2.1667, A 0.000, B 0.000, C 0.000 }
gfCNCPoint2[5182] = {X 332.5202, Y 4.0189, Z -2.1667, A 0.000, B 0.000, C 0.000 }
gfCNCPoint2[5183] = {X 334.0183, Y 3.1810, Z -2.1667, A 0.000, B 0.000, C 0.000 }
gfCNCPoint2[5184] = {X 335.5645, Y 2.4355, Z -2.1667, A 0.000, B 0.000, C 0.000 }
gfCNCPoint2[5185] = {X 337.6942, Y 1.5715, Z -2.1667, A 0.000, B 0.000, C 0.000 }
gfCNCPoint2[5186] = {X 339.8914, Y 0.8975, Z -2.1667, A 0.000, B 0.000, C 0.000 }
gfCNCPoint2[5187] = {X 342.1393, Y 0.4186, Z -2.1667, A 0.000, B 0.000, C 0.000 }
gfCNCPoint2[5188] = {X 344.4204, Y 0.1385, Z -2.1667, A 0.000, B 0.000, C 0.000 }
gfCNCPoint2[5189] = {X 346.7174, Y 0.0594, Z -2.1667, A 0.000, B 0.000, C 0.000 }
gfCNCPoint2[5190] = {X 349.0124, Y 0.1819, Z -2.1667, A 0.000, B 0.000, C 0.000 }
gfCNCPoint2[5191] = {X 351.2878, Y 0.5051, Z -2.1667, A 0.000, B 0.000, C 0.000 }
gfCNCPoint2[5192] = {X 351.5711, Y 0.5575, Z -2.1667, A 0.000, B 0.000, C 0.000 }
gfCNCPoint2[5193] = {X 352.2988, Y -3.3757, Z -2.1667, A 0.000, B 0.000, C 0.000 }
gfCNCPoint2[5194] = {X 351.5566, Y 0.6362, Z -2.1667, A 0.000, B 0.000, C 0.000 }
gfCNCPoint2[5195] = {X 351.8384, Y 0.6883, Z -2.1667, A 0.000, B 0.000, C 0.000 }
gfCNCPoint2[5196] = {X 353.7581, Y 1.1707, Z -2.1667, A 0.000, B 0.000, C 0.000 }
gfCNCPoint2[5197] = {X 355.6234, Y 1.8328, Z -2.1667, A 0.000, B 0.000, C 0.000 }
gfCNCPoint2[5198] = {X 357.4176, Y 2.6687, Z -2.1667, A 0.000, B 0.000, C 0.000 }
gfCNCPoint2[5199] = {X 359.1245, Y 3.6707, Z -2.1667, A 0.000, B 0.000, C 0.000 }
gfCNCPoint2[5200] = {X 360.7288, Y 4.8300, Z -2.1667, A 0.000, B 0.000, C 0.000 }
gfCNCPoint2[5201] = {X 362.2160, Y 6.1361, Z -2.1667, A 0.000, B 0.000, C 0.000 }
gfCNCPoint2[5202] = {X 363.5728, Y 7.5773, Z -2.1667, A 0.000, B 0.000, C 0.000 }
gfCNCPoint2[5203] = {X 365.0318, Y 9.4602, Z -2.1667, A 0.000, B 0.000, C 0.000 }
gfCNCPoint2[5204] = {X 366.3016, Y 11.4756, Z -2.1667, A 0.000, B 0.000, C 0.000 }
gfCNCPoint2[5205] = {X 367.3702, Y 13.6045, Z -2.1667, A 0.000, B 0.000, C 0.000 }
gfCNCPoint2[5206] = {X 368.2274, Y 15.8270, Z -2.1667, A 0.000, B 0.000, C 0.000 }
gfCNCPoint2[5207] = {X 368.8654, Y 18.1220, Z -2.1667, A 0.000, B 0.000, C 0.000 }
gfCNCPoint2[5208] = {X 369.3428, Y 20.7415, Z -2.1667, A 0.000, B 0.000, C 0.000 }
gfCNCPoint2[5209] = {X 369.5971, Y 23.3920, Z -2.1667, A 0.000, B 0.000, C 0.000 }
gfCNCPoint2[5210] = {X 369.6265, Y 26.0545, Z -2.1667, A 0.000, B 0.000, C 0.000 }
gfCNCPoint2[5211] = {X 369.4307, Y 28.7099, Z -2.1667, A 0.000, B 0.000, C 0.000 }
gfCNCPoint2[5212] = {X 369.0112, Y 31.3393, Z -2.1667, A 0.000, B 0.000, C 0.000 }
gfCNCPoint2[5213] = {X 368.4908, Y 33.4302, Z -2.1667, A 0.000, B 0.000, C 0.000 }
gfCNCPoint2[5214] = {X 367.7875, Y 35.4669, Z -2.1667, A 0.000, B 0.000, C 0.000 }
gfCNCPoint2[5215] = {X 366.9071, Y 37.4335, Z -2.1667, A 0.000, B 0.000, C 0.000 }
gfCNCPoint2[5216] = {X 365.8562, Y 39.3146, Z -2.1667, A 0.000, B 0.000, C 0.000 }
gfCNCPoint2[5217] = {X 364.6432, Y 41.0955, Z -2.1667, A 0.000, B 0.000, C 0.000 }
gfCNCPoint2[5218] = {X 363.4252, Y 42.5965, Z -2.1667, A 0.000, B 0.000, C 0.000 }
gfCNCPoint2[5219] = {X 362.0803, Y 43.9849, Z -2.1667, A 0.000, B 0.000, C 0.000 }
gfCNCPoint2[5220] = {X 360.6188, Y 45.2500, Z -2.1667, A 0.000, B 0.000, C 0.000 }
gfCNCPoint2[5221] = {X 359.0520, Y 46.3820, Z -2.1667, A 0.000, B 0.000, C 0.000 }
gfCNCPoint2[5222] = {X 357.3920, Y 47.3724, Z -2.1667, A 0.000, B 0.000, C 0.000 }
gfCNCPoint2[5223] = {X 355.4451, Y 48.2564, Z -2.1667, A 0.000, B 0.000, C 0.000 }
gfCNCPoint2[5224] = {X 353.4230, Y 48.9513, Z -2.1667, A 0.000, B 0.000, C 0.000 }
gfCNCPoint2[5225] = {X 351.3440, Y 49.4509, Z -2.1667, A 0.000, B 0.000, C 0.000 }
gfCNCPoint2[5226] = {X 349.2269, Y 49.7507, Z -2.1667, A 0.000, B 0.000, C 0.000 }
gfCNCPoint2[5227] = {X 347.0909, Y 49.8479, Z -2.1667, A 0.000, B 0.000, C 0.000 }
gfCNCPoint2[5228] = {X 345.0381, Y 49.8135, Z -2.1667, A 0.000, B 0.000, C 0.000 }
gfCNCPoint2[5229] = {X 342.9961, Y 49.6011, Z -2.1667, A 0.000, B 0.000, C 0.000 }
gfCNCPoint2[5230] = {X 340.9801, Y 49.2124, Z -2.1667, A 0.000, B 0.000, C 0.000 }
gfCNCPoint2[5231] = {X 339.0055, Y 48.6504, Z -2.1667, A 0.000, B 0.000, C 0.000 }
gfCNCPoint2[5232] = {X 337.0871, Y 47.9191, Z -2.1667, A 0.000, B 0.000, C 0.000 }
gfCNCPoint2[5233] = {X 335.2393, Y 47.0242, Z -2.1667, A 0.000, B 0.000, C 0.000 }
gfCNCPoint2[5234] = {X 333.6469, Y 46.0386, Z -2.1667, A 0.000, B 0.000, C 0.000 }
gfCNCPoint2[5235] = {X 332.1365, Y 44.9314, Z -2.1667, A 0.000, B 0.000, C 0.000 }
gfCNCPoint2[5236] = {X 330.7174, Y 43.7094, Z -2.1667, A 0.000, B 0.000, C 0.000 }
gfCNCPoint2[5237] = {X 329.7932, Y 43.7230, Z -2.1667, A 0.000, B 0.000, C 0.000 }
gfCNCPoint2[5238] = {X 328.8888, Y 43.5323, Z -2.1667, A 0.000, B 0.000, C 0.000 }
gfCNCPoint2[5239] = {X 328.0488, Y 43.1465, Z -2.1667, A 0.000, B 0.000, C 0.000 }
gfCNCPoint2[5240] = {X 327.3148, Y 42.5847, Z -2.1667, A 0.000, B 0.000, C 0.000 }
gfCNCPoint2[5241] = {X 326.6925, Y 41.9780, Z -2.1667, A 0.000, B 0.000, C 0.000 }
gfCNCPoint2[5242] = {X 326.0873, Y 41.2331, Z -2.1667, A 0.000, B 0.000, C 0.000 }
gfCNCPoint2[5243] = {X 325.6690, Y 40.3693, Z -2.1667, A 0.000, B 0.000, C 0.000 }
gfCNCPoint2[5244] = {X 325.4597, Y 39.4326, Z -2.1667, A 0.000, B 0.000, C 0.000 }
gfCNCPoint2[5245] = {X 325.4707, Y 38.4730, Z -2.1667, A 0.000, B 0.000, C 0.000 }
gfCNCPoint2[5246] = {X 325.7013, Y 37.5413, Z -2.1667, A 0.000, B 0.000, C 0.000 }
gfCNCPoint2[5247] = {X 326.1392, Y 36.6874, Z -2.1667, A 0.000, B 0.000, C 0.000 }
gfCNCPoint2[5248] = {X 330.3969, Y 30.3216, Z -2.1667, A 0.000, B 0.000, C 0.000 }
gfCNCPoint2[5249] = {X 330.9792, Y 29.6411, Z -2.1667, A 0.000, B 0.000, C 0.000 }
gfCNCPoint2[5250] = {X 331.6937, Y 29.1010, Z -2.1667, A 0.000, B 0.000, C 0.000 }
gfCNCPoint2[5251] = {X 332.5073, Y 28.7264, Z -2.1667, A 0.000, B 0.000, C 0.000 }
gfCNCPoint2[5252] = {X 333.3822, Y 28.5346, Z -2.1667, A 0.000, B 0.000, C 0.000 }
gfCNCPoint2[5253] = {X 334.2779, Y 28.5345, Z -2.1667, A 0.000, B 0.000, C 0.000 }
gfCNCPoint2[5254] = {X 335.1528, Y 28.7261, Z -2.1667, A 0.000, B 0.000, C 0.000 }
gfCNCPoint2[5255] = {X 335.9664, Y 29.1006, Z -2.1667, A 0.000, B 0.000, C 0.000 }
gfCNCPoint2[5256] = {X 336.6810, Y 29.6405, Z -2.1667, A 0.000, B 0.000, C 0.000 }
gfCNCPoint2[5257] = {X 337.3163, Y 30.2523, Z -2.1667, A 0.000, B 0.000, C 0.000 }
gfCNCPoint2[5258] = {X 337.8308, Y 30.8659, Z -2.1667, A 0.000, B 0.000, C 0.000 }
gfCNCPoint2[5259] = {X 338.2182, Y 31.5666, Z -2.1667, A 0.000, B 0.000, C 0.000 }
gfCNCPoint2[5260] = {X 338.4642, Y 32.3287, Z -2.1667, A 0.000, B 0.000, C 0.000 }
gfCNCPoint2[5261] = {X 338.5597, Y 33.1237, Z -2.1667, A 0.000, B 0.000, C 0.000 }
gfCNCPoint2[5262] = {X 338.5011, Y 33.9223, Z -2.1667, A 0.000, B 0.000, C 0.000 }
gfCNCPoint2[5263] = {X 339.2993, Y 34.6502, Z -2.1667, A 0.000, B 0.000, C 0.000 }
gfCNCPoint2[5264] = {X 340.1350, Y 35.3347, Z -2.1667, A 0.000, B 0.000, C 0.000 }
gfCNCPoint2[5265] = {X 341.4515, Y 36.1997, Z -2.1667, A 0.000, B 0.000, C 0.000 }
gfCNCPoint2[5266] = {X 342.8801, Y 36.8635, Z -2.1667, A 0.000, B 0.000, C 0.000 }
gfCNCPoint2[5267] = {X 344.3902, Y 37.3119, Z -2.1667, A 0.000, B 0.000, C 0.000 }
gfCNCPoint2[5268] = {X 345.9496, Y 37.5353, Z -2.1667, A 0.000, B 0.000, C 0.000 }
gfCNCPoint2[5269] = {X 347.5248, Y 37.5290, Z -2.1667, A 0.000, B 0.000, C 0.000 }
gfCNCPoint2[5270] = {X 348.7033, Y 37.3903, Z -2.1667, A 0.000, B 0.000, C 0.000 }
gfCNCPoint2[5271] = {X 349.8535, Y 37.0987, Z -2.1667, A 0.000, B 0.000, C 0.000 }
gfCNCPoint2[5272] = {X 350.9557, Y 36.6593, Z -2.1667, A 0.000, B 0.000, C 0.000 }
gfCNCPoint2[5273] = {X 351.9910, Y 36.0796, Z -2.1667, A 0.000, B 0.000, C 0.000 }
gfCNCPoint2[5274] = {X 352.9416, Y 35.3694, Z -2.1667, A 0.000, B 0.000, C 0.000 }
gfCNCPoint2[5275] = {X 354.1074, Y 34.2343, Z -2.1667, A 0.000, B 0.000, C 0.000 }
gfCNCPoint2[5276] = {X 355.1164, Y 32.9578, Z -2.1667, A 0.000, B 0.000, C 0.000 }
gfCNCPoint2[5277] = {X 355.9516, Y 31.5614, Z -2.1667, A 0.000, B 0.000, C 0.000 }
gfCNCPoint2[5278] = {X 356.5990, Y 30.0686, Z -2.1667, A 0.000, B 0.000, C 0.000 }
gfCNCPoint2[5279] = {X 357.0476, Y 28.5046, Z -2.1667, A 0.000, B 0.000, C 0.000 }
gfCNCPoint2[5280] = {X 357.3234, Y 26.8012, Z -2.1667, A 0.000, B 0.000, C 0.000 }
gfCNCPoint2[5281] = {X 357.4357, Y 25.0793, Z -2.1667, A 0.000, B 0.000, C 0.000 }
gfCNCPoint2[5282] = {X 357.3836, Y 23.3545, Z -2.1667, A 0.000, B 0.000, C 0.000 }
gfCNCPoint2[5283] = {X 357.1675, Y 21.6425, Z -2.1667, A 0.000, B 0.000, C 0.000 }
gfCNCPoint2[5284] = {X 356.8267, Y 20.1740, Z -2.1667, A 0.000, B 0.000, C 0.000 }
gfCNCPoint2[5285] = {X 356.3068, Y 18.7589, Z -2.1667, A 0.000, B 0.000, C 0.000 }
gfCNCPoint2[5286] = {X 355.6158, Y 17.4189, Z -2.1667, A 0.000, B 0.000, C 0.000 }
gfCNCPoint2[5287] = {X 354.7644, Y 16.1748, Z -2.1667, A 0.000, B 0.000, C 0.000 }
gfCNCPoint2[5288] = {X 353.8631, Y 15.1697, Z -2.1667, A 0.000, B 0.000, C 0.000 }
gfCNCPoint2[5289] = {X 352.8271, Y 14.3040, Z -2.1667, A 0.000, B 0.000, C 0.000 }
gfCNCPoint2[5290] = {X 351.6778, Y 13.5957, Z -2.1667, A 0.000, B 0.000, C 0.000 }
gfCNCPoint2[5291] = {X 350.4389, Y 13.0593, Z -2.1667, A 0.000, B 0.000, C 0.000 }
gfCNCPoint2[5292] = {X 349.1359, Y 12.7059, Z -2.1667, A 0.000, B 0.000, C 0.000 }
gfCNCPoint2[5293] = {X 347.5975, Y 12.5006, Z -2.1667, A 0.000, B 0.000, C 0.000 }
gfCNCPoint2[5294] = {X 346.0456, Y 12.4726, Z -2.1667, A 0.000, B 0.000, C 0.000 }
gfCNCPoint2[5295] = {X 344.5008, Y 12.6224, Z -2.1667, A 0.000, B 0.000, C 0.000 }
gfCNCPoint2[5296] = {X 342.9832, Y 12.9479, Z -2.1667, A 0.000, B 0.000, C 0.000 }
gfCNCPoint2[5297] = {X 341.5128, Y 13.4449, Z -2.1667, A 0.000, B 0.000, C 0.000 }
gfCNCPoint2[5298] = {X 340.1090, Y 14.1069, Z -2.1667, A 0.000, B 0.000, C 0.000 }
gfCNCPoint2[5299] = {X 338.7901, Y 14.9251, Z -2.1667, A 0.000, B 0.000, C 0.000 }
gfCNCPoint2[5300] = {X 338.7679, Y 15.7566, Z -2.1667, A 0.000, B 0.000, C 0.000 }
gfCNCPoint2[5301] = {X 338.5808, Y 16.5671, Z -2.1667, A 0.000, B 0.000, C 0.000 }
gfCNCPoint2[5302] = {X 338.2362, Y 17.3242, Z -2.1667, A 0.000, B 0.000, C 0.000 }
gfCNCPoint2[5303] = {X 337.7479, Y 17.9976, Z -2.1667, A 0.000, B 0.000, C 0.000 }
gfCNCPoint2[5304] = {X 337.1353, Y 18.5603, Z -2.1667, A 0.000, B 0.000, C 0.000 }
gfCNCPoint2[5305] = {X 336.4209, Y 19.0861, Z -2.1667, A 0.000, B 0.000, C 0.000 }
gfCNCPoint2[5306] = {X 335.6353, Y 19.5283, Z -2.1667, A 0.000, B 0.000, C 0.000 }
gfCNCPoint2[5307] = {X 334.7729, Y 19.7908, Z -2.1667, A 0.000, B 0.000, C 0.000 }
gfCNCPoint2[5308] = {X 333.8742, Y 19.8614, Z -2.1667, A 0.000, B 0.000, C 0.000 }
gfCNCPoint2[5309] = {X 332.9814, Y 19.7367, Z -2.1667, A 0.000, B 0.000, C 0.000 }
gfCNCPoint2[5310] = {X 332.1364, Y 19.4226, Z -2.1667, A 0.000, B 0.000, C 0.000 }
gfCNCPoint2[5311] = {X 331.3789, Y 18.9339, Z -2.1667, A 0.000, B 0.000, C 0.000 }
gfCNCPoint2[5312] = {X 330.7445, Y 18.2934, Z -2.1667, A 0.000, B 0.000, C 0.000 }
gfCNCPoint2[5313] = {X 330.2630, Y 17.5314, Z -2.1667, A 0.000, B 0.000, C 0.000 }
gfCNCPoint2[5314] = {X 326.7381, Y 10.2803, Z -2.1667, A 0.000, B 0.000, C 0.000 }
gfCNCPoint2[5315] = {X 326.4156, Y 9.3505, Z -2.1667, A 0.000, B 0.000, C 0.000 }
gfCNCPoint2[5316] = {X 326.3205, Y 8.3711, Z -2.1667, A 0.000, B 0.000, C 0.000 }
gfCNCPoint2[5317] = {X 326.4581, Y 7.3967, Z -2.1667, A 0.000, B 0.000, C 0.000 }
gfCNCPoint2[5318] = {X 326.8207, Y 6.4819, Z -2.1667, A 0.000, B 0.000, C 0.000 }
gfCNCPoint2[5319] = {X 327.3881, Y 5.6778, Z -2.1667, A 0.000, B 0.000, C 0.000 }
gfCNCPoint2[5320] = {X 328.1285, Y 5.0296, Z -2.1667, A 0.000, B 0.000, C 0.000 }
gfCNCPoint2[5321] = {X 328.7983, Y 4.5709, Z -2.1667, A 0.000, B 0.000, C 0.000 }
gfCNCPoint2[5322] = {X 329.6634, Y 4.1256, Z -2.1667, A 0.000, B 0.000, C 0.000 }
gfCNCPoint2[5323] = {X 330.6083, Y 3.8934, Z -2.1667, A 0.000, B 0.000, C 0.000 }
gfCNCPoint2[5324] = {X 331.5812, Y 3.8870, Z -2.1667, A 0.000, B 0.000, C 0.000 }
gfCNCPoint2[5325] = {X 332.5291, Y 4.1069, Z -2.1667, A 0.000, B 0.000, C 0.000 }
gfCNCPoint2[5326] = {X 334.0387, Y 3.2605, Z -2.1667, A 0.000, B 0.000, C 0.000 }
gfCNCPoint2[5327] = {X 335.5974, Y 2.5084, Z -2.1667, A 0.000, B 0.000, C 0.000 }
gfCNCPoint2[5328] = {X 337.7207, Y 1.6470, Z -2.1667, A 0.000, B 0.000, C 0.000 }
gfCNCPoint2[5329] = {X 339.9113, Y 0.9750, Z -2.1667, A 0.000, B 0.000, C 0.000 }
gfCNCPoint2[5330] = {X 342.1523, Y 0.4975, Z -2.1667, A 0.000, B 0.000, C 0.000 }
gfCNCPoint2[5331] = {X 344.4266, Y 0.2183, Z -2.1667, A 0.000, B 0.000, C 0.000 }
gfCNCPoint2[5332] = {X 346.7165, Y 0.1394, Z -2.1667, A 0.000, B 0.000, C 0.000 }
gfCNCPoint2[5333] = {X 349.0046, Y 0.2616, Z -2.1667, A 0.000, B 0.000, C 0.000 }
gfCNCPoint2[5334] = {X 351.2732, Y 0.5838, Z -2.1667, A 0.000, B 0.000, C 0.000 }
gfCNCPoint2[5335] = {X 351.5566, Y 0.6362, Z -2.1667, A 0.000, B 0.000, C 0.000 }
gfCNCPoint2[5336] = {X 352.2842, Y -3.2971, Z -2.1667, A 0.000, B 0.000, C 0.000 }
gfCNCPoint2[5337] = {X 351.5420, Y 0.7148, Z -2.1667, A 0.000, B 0.000, C 0.000 }
gfCNCPoint2[5338] = {X 351.8233, Y 0.7669, Z -2.1667, A 0.000, B 0.000, C 0.000 }
gfCNCPoint2[5339] = {X 353.7354, Y 1.2474, Z -2.1667, A 0.000, B 0.000, C 0.000 }
gfCNCPoint2[5340] = {X 355.5935, Y 1.9070, Z -2.1667, A 0.000, B 0.000, C 0.000 }
gfCNCPoint2[5341] = {X 357.3807, Y 2.7397, Z -2.1667, A 0.000, B 0.000, C 0.000 }
gfCNCPoint2[5342] = {X 359.0810, Y 3.7379, Z -2.1667, A 0.000, B 0.000, C 0.000 }
gfCNCPoint2[5343] = {X 360.6790, Y 4.8927, Z -2.1667, A 0.000, B 0.000, C 0.000 }
gfCNCPoint2[5344] = {X 362.1605, Y 6.1937, Z -2.1667, A 0.000, B 0.000, C 0.000 }
gfCNCPoint2[5345] = {X 363.5120, Y 7.6293, Z -2.1667, A 0.000, B 0.000, C 0.000 }
gfCNCPoint2[5346] = {X 364.9663, Y 9.5061, Z -2.1667, A 0.000, B 0.000, C 0.000 }
gfCNCPoint2[5347] = {X 366.2319, Y 11.5149, Z -2.1667, A 0.000, B 0.000, C 0.000 }
gfCNCPoint2[5348] = {X 367.2970, Y 13.6369, Z -2.1667, A 0.000, B 0.000, C 0.000 }
gfCNCPoint2[5349] = {X 368.1515, Y 15.8521, Z -2.1667, A 0.000, B 0.000, C 0.000 }
gfCNCPoint2[5350] = {X 368.7873, Y 18.1397, Z -2.1667, A 0.000, B 0.000, C 0.000 }
gfCNCPoint2[5351] = {X 369.2636, Y 20.7525, Z -2.1667, A 0.000, B 0.000, C 0.000 }
gfCNCPoint2[5352] = {X 369.5173, Y 23.3962, Z -2.1667, A 0.000, B 0.000, C 0.000 }
gfCNCPoint2[5353] = {X 369.5466, Y 26.0519, Z -2.1667, A 0.000, B 0.000, C 0.000 }
gfCNCPoint2[5354] = {X 369.3513, Y 28.7006, Z -2.1667, A 0.000, B 0.000, C 0.000 }
gfCNCPoint2[5355] = {X 368.9328, Y 31.3234, Z -2.1667, A 0.000, B 0.000, C 0.000 }
gfCNCPoint2[5356] = {X 368.4141, Y 33.4074, Z -2.1667, A 0.000, B 0.000, C 0.000 }
gfCNCPoint2[5357] = {X 367.7131, Y 35.4375, Z -2.1667, A 0.000, B 0.000, C 0.000 }
gfCNCPoint2[5358] = {X 366.8355, Y 37.3977, Z -2.1667, A 0.000, B 0.000, C 0.000 }
gfCNCPoint2[5359] = {X 365.7881, Y 39.2726, Z -2.1667, A 0.000, B 0.000, C 0.000 }
gfCNCPoint2[5360] = {X 364.5791, Y 41.0476, Z -2.1667, A 0.000, B 0.000, C 0.000 }
gfCNCPoint2[5361] = {X 363.3656, Y 42.5431, Z -2.1667, A 0.000, B 0.000, C 0.000 }
gfCNCPoint2[5362] = {X 362.0257, Y 43.9264, Z -2.1667, A 0.000, B 0.000, C 0.000 }
gfCNCPoint2[5363] = {X 360.5696, Y 45.1869, Z -2.1667, A 0.000, B 0.000, C 0.000 }
gfCNCPoint2[5364] = {X 359.0086, Y 46.3148, Z -2.1667, A 0.000, B 0.000, C 0.000 }
gfCNCPoint2[5365] = {X 357.3547, Y 47.3015, Z -2.1667, A 0.000, B 0.000, C 0.000 }
gfCNCPoint2[5366] = {X 355.4147, Y 48.1823, Z -2.1667, A 0.000, B 0.000, C 0.000 }
gfCNCPoint2[5367] = {X 353.3997, Y 48.8748, Z -2.1667, A 0.000, B 0.000, C 0.000 }
gfCNCPoint2[5368] = {X 351.3280, Y 49.3725, Z -2.1667, A 0.000, B 0.000, C 0.000 }
gfCNCPoint2[5369] = {X 349.2184, Y 49.6712, Z -2.1667, A 0.000, B 0.000, C 0.000 }
gfCNCPoint2[5370] = {X 347.0899, Y 49.7679, Z -2.1667, A 0.000, B 0.000, C 0.000 }
gfCNCPoint2[5371] = {X 345.0440, Y 49.7337, Z -2.1667, A 0.000, B 0.000, C 0.000 }
gfCNCPoint2[5372] = {X 343.0088, Y 49.5221, Z -2.1667, A 0.000, B 0.000, C 0.000 }
gfCNCPoint2[5373] = {X 340.9996, Y 49.1348, Z -2.1667, A 0.000, B 0.000, C 0.000 }
gfCNCPoint2[5374] = {X 339.0316, Y 48.5747, Z -2.1667, A 0.000, B 0.000, C 0.000 }
gfCNCPoint2[5375] = {X 337.1196, Y 47.8460, Z -2.1667, A 0.000, B 0.000, C 0.000 }
gfCNCPoint2[5376] = {X 335.2780, Y 46.9542, Z -2.1667, A 0.000, B 0.000, C 0.000 }
gfCNCPoint2[5377] = {X 333.6808, Y 45.9650, Z -2.1667, A 0.000, B 0.000, C 0.000 }
gfCNCPoint2[5378] = {X 332.1664, Y 44.8530, Z -2.1667, A 0.000, B 0.000, C 0.000 }
gfCNCPoint2[5379] = {X 330.7444, Y 43.6252, Z -2.1667, A 0.000, B 0.000, C 0.000 }
gfCNCPoint2[5380] = {X 329.8288, Y 43.6460, Z -2.1667, A 0.000, B 0.000, C 0.000 }
gfCNCPoint2[5381] = {X 328.9316, Y 43.4621, Z -2.1667, A 0.000, B 0.000, C 0.000 }
gfCNCPoint2[5382] = {X 328.0981, Y 43.0827, Z -2.1667, A 0.000, B 0.000, C 0.000 }
gfCNCPoint2[5383] = {X 327.3701, Y 42.5270, Z -2.1667, A 0.000, B 0.000, C 0.000 }
gfCNCPoint2[5384] = {X 326.7483, Y 41.9207, Z -2.1667, A 0.000, B 0.000, C 0.000 }
gfCNCPoint2[5385] = {X 326.1548, Y 41.1901, Z -2.1667, A 0.000, B 0.000, C 0.000 }
gfCNCPoint2[5386] = {X 325.7445, Y 40.3430, Z -2.1667, A 0.000, B 0.000, C 0.000 }
gfCNCPoint2[5387] = {X 325.5393, Y 39.4243, Z -2.1667, A 0.000, B 0.000, C 0.000 }
gfCNCPoint2[5388] = {X 325.5500, Y 38.4831, Z -2.1667, A 0.000, B 0.000, C 0.000 }
gfCNCPoint2[5389] = {X 325.7762, Y 37.5694, Z -2.1667, A 0.000, B 0.000, C 0.000 }
gfCNCPoint2[5390] = {X 326.2057, Y 36.7318, Z -2.1667, A 0.000, B 0.000, C 0.000 }
gfCNCPoint2[5391] = {X 330.4629, Y 30.3668, Z -2.1667, A 0.000, B 0.000, C 0.000 }
gfCNCPoint2[5392] = {X 331.0340, Y 29.6994, Z -2.1667, A 0.000, B 0.000, C 0.000 }
gfCNCPoint2[5393] = {X 331.7347, Y 29.1697, Z -2.1667, A 0.000, B 0.000, C 0.000 }
gfCNCPoint2[5394] = {X 332.5326, Y 28.8023, Z -2.1667, A 0.000, B 0.000, C 0.000 }
gfCNCPoint2[5395] = {X 333.3906, Y 28.6141, Z -2.1667, A 0.000, B 0.000, C 0.000 }
gfCNCPoint2[5396] = {X 334.2690, Y 28.6140, Z -2.1667, A 0.000, B 0.000, C 0.000 }
gfCNCPoint2[5397] = {X 335.1270, Y 28.8018, Z -2.1667, A 0.000, B 0.000, C 0.000 }
gfCNCPoint2[5398] = {X 335.9250, Y 29.1690, Z -2.1667, A 0.000, B 0.000, C 0.000 }
gfCNCPoint2[5399] = {X 336.6259, Y 29.6985, Z -2.1667, A 0.000, B 0.000, C 0.000 }
gfCNCPoint2[5400] = {X 337.2602, Y 30.3094, Z -2.1667, A 0.000, B 0.000, C 0.000 }
gfCNCPoint2[5401] = {X 337.7696, Y 30.9181, Z -2.1667, A 0.000, B 0.000, C 0.000 }
gfCNCPoint2[5402] = {X 338.1515, Y 31.6139, Z -2.1667, A 0.000, B 0.000, C 0.000 }
gfCNCPoint2[5403] = {X 338.3914, Y 32.3705, Z -2.1667, A 0.000, B 0.000, C 0.000 }
gfCNCPoint2[5404] = {X 338.4804, Y 33.1593, Z -2.1667, A 0.000, B 0.000, C 0.000 }
gfCNCPoint2[5405] = {X 338.4149, Y 33.9503, Z -2.1667, A 0.000, B 0.000, C 0.000 }
gfCNCPoint2[5406] = {X 339.2309, Y 34.6968, Z -2.1667, A 0.000, B 0.000, C 0.000 }
gfCNCPoint2[5407] = {X 340.0861, Y 35.3980, Z -2.1667, A 0.000, B 0.000, C 0.000 }
gfCNCPoint2[5408] = {X 341.4123, Y 36.2694, Z -2.1667, A 0.000, B 0.000, C 0.000 }
gfCNCPoint2[5409] = {X 342.8513, Y 36.9381, Z -2.1667, A 0.000, B 0.000, C 0.000 }
gfCNCPoint2[5410] = {X 344.3724, Y 37.3899, Z -2.1667, A 0.000, B 0.000, C 0.000 }
gfCNCPoint2[5411] = {X 345.9432, Y 37.6151, Z -2.1667, A 0.000, B 0.000, C 0.000 }
gfCNCPoint2[5412] = {X 347.5300, Y 37.6088, Z -2.1667, A 0.000, B 0.000, C 0.000 }
gfCNCPoint2[5413] = {X 348.7186, Y 37.4688, Z -2.1667, A 0.000, B 0.000, C 0.000 }
gfCNCPoint2[5414] = {X 349.8788, Y 37.1746, Z -2.1667, A 0.000, B 0.000, C 0.000 }
gfCNCPoint2[5415] = {X 350.9905, Y 36.7313, Z -2.1667, A 0.000, B 0.000, C 0.000 }
gfCNCPoint2[5416] = {X 352.0348, Y 36.1465, Z -2.1667, A 0.000, B 0.000, C 0.000 }
gfCNCPoint2[5417] = {X 352.9936, Y 35.4302, Z -2.1667, A 0.000, B 0.000, C 0.000 }
gfCNCPoint2[5418] = {X 354.1669, Y 34.2878, Z -2.1667, A 0.000, B 0.000, C 0.000 }
gfCNCPoint2[5419] = {X 355.1823, Y 33.0032, Z -2.1667, A 0.000, B 0.000, C 0.000 }
gfCNCPoint2[5420] = {X 356.0228, Y 31.5978, Z -2.1667, A 0.000, B 0.000, C 0.000 }
gfCNCPoint2[5421] = {X 356.6743, Y 30.0954, Z -2.1667, A 0.000, B 0.000, C 0.000 }
gfCNCPoint2[5422] = {X 357.1258, Y 28.5214, Z -2.1667, A 0.000, B 0.000, C 0.000 }
gfCNCPoint2[5423] = {X 357.4028, Y 26.8104, Z -2.1667, A 0.000, B 0.000, C 0.000 }
gfCNCPoint2[5424] = {X 357.5157, Y 25.0808, Z -2.1667, A 0.000, B 0.000, C 0.000 }
gfCNCPoint2[5425] = {X 357.4634, Y 23.3484, Z -2.1667, A 0.000, B 0.000, C 0.000 }
gfCNCPoint2[5426] = {X 357.2463, Y 21.6288, Z -2.1667, A 0.000, B 0.000, C 0.000 }
gfCNCPoint2[5427] = {X 356.9032, Y 20.1507, Z -2.1667, A 0.000, B 0.000, C 0.000 }
gfCNCPoint2[5428] = {X 356.3799, Y 18.7264, Z -2.1667, A 0.000, B 0.000, C 0.000 }
gfCNCPoint2[5429] = {X 355.6845, Y 17.3778, Z -2.1667, A 0.000, B 0.000, C 0.000 }
gfCNCPoint2[5430] = {X 354.8275, Y 16.1256, Z -2.1667, A 0.000, B 0.000, C 0.000 }
gfCNCPoint2[5431] = {X 353.9185, Y 15.1120, Z -2.1667, A 0.000, B 0.000, C 0.000 }
gfCNCPoint2[5432] = {X 352.8737, Y 14.2390, Z -2.1667, A 0.000, B 0.000, C 0.000 }
gfCNCPoint2[5433] = {X 351.7146, Y 13.5247, Z -2.1667, A 0.000, B 0.000, C 0.000 }
gfCNCPoint2[5434] = {X 350.4652, Y 12.9838, Z -2.1667, A 0.000, B 0.000, C 0.000 }
gfCNCPoint2[5435] = {X 349.1511, Y 12.6274, Z -2.1667, A 0.000, B 0.000, C 0.000 }
gfCNCPoint2[5436] = {X 347.5972, Y 12.4203, Z -2.1667, A 0.000, B 0.000, C 0.000 }
gfCNCPoint2[5437] = {X 346.0297, Y 12.3932, Z -2.1667, A 0.000, B 0.000, C 0.000 }
gfCNCPoint2[5438] = {X 344.4695, Y 12.5463, Z -2.1667, A 0.000, B 0.000, C 0.000 }
gfCNCPoint2[5439] = {X 342.9372, Y 12.8776, Z -2.1667, A 0.000, B 0.000, C 0.000 }
gfCNCPoint2[5440] = {X 341.4531, Y 13.3827, Z -2.1667, A 0.000, B 0.000, C 0.000 }
gfCNCPoint2[5441] = {X 340.0369, Y 14.0551, Z -2.1667, A 0.000, B 0.000, C 0.000 }
gfCNCPoint2[5442] = {X 338.7073, Y 14.8856, Z -2.1667, A 0.000, B 0.000, C 0.000 }
gfCNCPoint2[5443] = {X 338.7152, Y 15.0049, Z -2.1667, A 0.000, B 0.000, C 0.000 }
gfCNCPoint2[5444] = {X 338.6808, Y 15.8052, Z -2.1667, A 0.000, B 0.000, C 0.000 }
gfCNCPoint2[5445] = {X 338.4907, Y 16.5835, Z -2.1667, A 0.000, B 0.000, C 0.000 }
gfCNCPoint2[5446] = {X 338.1522, Y 17.3095, Z -2.1667, A 0.000, B 0.000, C 0.000 }
gfCNCPoint2[5447] = {X 337.6783, Y 17.9554, Z -2.1667, A 0.000, B 0.000, C 0.000 }
gfCNCPoint2[5448] = {X 337.0874, Y 18.4963, Z -2.1667, A 0.000, B 0.000, C 0.000 }
gfCNCPoint2[5449] = {X 336.3744, Y 19.0211, Z -2.1667, A 0.000, B 0.000, C 0.000 }
gfCNCPoint2[5450] = {X 335.6039, Y 19.4547, Z -2.1667, A 0.000, B 0.000, C 0.000 }
gfCNCPoint2[5451] = {X 334.7580, Y 19.7122, Z -2.1667, A 0.000, B 0.000, C 0.000 }
gfCNCPoint2[5452] = {X 333.8766, Y 19.7814, Z -2.1667, A 0.000, B 0.000, C 0.000 }
gfCNCPoint2[5453] = {X 333.0010, Y 19.6592, Z -2.1667, A 0.000, B 0.000, C 0.000 }
gfCNCPoint2[5454] = {X 332.1722, Y 19.3511, Z -2.1667, A 0.000, B 0.000, C 0.000 }
gfCNCPoint2[5455] = {X 331.4293, Y 18.8718, Z -2.1667, A 0.000, B 0.000, C 0.000 }
gfCNCPoint2[5456] = {X 330.8071, Y 18.2436, Z -2.1667, A 0.000, B 0.000, C 0.000 }
gfCNCPoint2[5457] = {X 330.3348, Y 17.4962, Z -2.1667, A 0.000, B 0.000, C 0.000 }
gfCNCPoint2[5458] = {X 326.8100, Y 10.2453, Z -2.1667, A 0.000, B 0.000, C 0.000 }
gfCNCPoint2[5459] = {X 326.4937, Y 9.3334, Z -2.1667, A 0.000, B 0.000, C 0.000 }
gfCNCPoint2[5460] = {X 326.4004, Y 8.3728, Z -2.1667, A 0.000, B 0.000, C 0.000 }
gfCNCPoint2[5461] = {X 326.5354, Y 7.4171, Z -2.1667, A 0.000, B 0.000, C 0.000 }
gfCNCPoint2[5462] = {X 326.8911, Y 6.5199, Z -2.1667, A 0.000, B 0.000, C 0.000 }
gfCNCPoint2[5463] = {X 327.4476, Y 5.7314, Z -2.1667, A 0.000, B 0.000, C 0.000 }
gfCNCPoint2[5464] = {X 328.1737, Y 5.0956, Z -2.1667, A 0.000, B 0.000, C 0.000 }
gfCNCPoint2[5465] = {X 328.8432, Y 4.6371, Z -2.1667, A 0.000, B 0.000, C 0.000 }
gfCNCPoint2[5466] = {X 329.7005, Y 4.1971, Z -2.1667, A 0.000, B 0.000, C 0.000 }
gfCNCPoint2[5467] = {X 330.6371, Y 3.9705, Z -2.1667, A 0.000, B 0.000, C 0.000 }
gfCNCPoint2[5468] = {X 331.6007, Y 3.9698, Z -2.1667, A 0.000, B 0.000, C 0.000 }
gfCNCPoint2[5469] = {X 332.5376, Y 4.1951, Z -2.1667, A 0.000, B 0.000, C 0.000 }
gfCNCPoint2[5470] = {X 334.0589, Y 3.3402, Z -2.1667, A 0.000, B 0.000, C 0.000 }
gfCNCPoint2[5471] = {X 335.6304, Y 2.5813, Z -2.1667, A 0.000, B 0.000, C 0.000 }
gfCNCPoint2[5472] = {X 337.7472, Y 1.7225, Z -2.1667, A 0.000, B 0.000, C 0.000 }
gfCNCPoint2[5473] = {X 339.9311, Y 1.0525, Z -2.1667, A 0.000, B 0.000, C 0.000 }
gfCNCPoint2[5474] = {X 342.1653, Y 0.5764, Z -2.1667, A 0.000, B 0.000, C 0.000 }
gfCNCPoint2[5475] = {X 344.4327, Y 0.2980, Z -2.1667, A 0.000, B 0.000, C 0.000 }
gfCNCPoint2[5476] = {X 346.7157, Y 0.2194, Z -2.1667, A 0.000, B 0.000, C 0.000 }
gfCNCPoint2[5477] = {X 348.9968, Y 0.3412, Z -2.1667, A 0.000, B 0.000, C 0.000 }
gfCNCPoint2[5478] = {X 351.2585, Y 0.6624, Z -2.1667, A 0.000, B 0.000, C 0.000 }
gfCNCPoint2[5479] = {X 351.5420, Y 0.7148, Z -2.1667, A 0.000, B 0.000, C 0.000 }
gfCNCPoint2[5480] = {X 352.2697, Y -3.2184, Z -2.1667, A 0.000, B 0.000, C 0.000 }
gfCNCPoint2[5481] = {X 351.5275, Y 0.7935, Z -2.1667, A 0.000, B 0.000, C 0.000 }
gfCNCPoint2[5482] = {X 351.8081, Y 0.8454, Z -2.1667, A 0.000, B 0.000, C 0.000 }
gfCNCPoint2[5483] = {X 353.7128, Y 1.3242, Z -2.1667, A 0.000, B 0.000, C 0.000 }
gfCNCPoint2[5484] = {X 355.5636, Y 1.9812, Z -2.1667, A 0.000, B 0.000, C 0.000 }
gfCNCPoint2[5485] = {X 357.3438, Y 2.8107, Z -2.1667, A 0.000, B 0.000, C 0.000 }
gfCNCPoint2[5486] = {X 359.0375, Y 3.8050, Z -2.1667, A 0.000, B 0.000, C 0.000 }
gfCNCPoint2[5487] = {X 360.6293, Y 4.9554, Z -2.1667, A 0.000, B 0.000, C 0.000 }
gfCNCPoint2[5488] = {X 362.1050, Y 6.2513, Z -2.1667, A 0.000, B 0.000, C 0.000 }
gfCNCPoint2[5489] = {X 363.4512, Y 7.6813, Z -2.1667, A 0.000, B 0.000, C 0.000 }
gfCNCPoint2[5490] = {X 364.9008, Y 9.5519, Z -2.1667, A 0.000, B 0.000, C 0.000 }
gfCNCPoint2[5491] = {X 366.1623, Y 11.5542, Z -2.1667, A 0.000, B 0.000, C 0.000 }
gfCNCPoint2[5492] = {X 367.2238, Y 13.6693, Z -2.1667, A 0.000, B 0.000, C 0.000 }
gfCNCPoint2[5493] = {X 368.0755, Y 15.8772, Z -2.1667, A 0.000, B 0.000, C 0.000 }
gfCNCPoint2[5494] = {X 368.7093, Y 18.1573, Z -2.1667, A 0.000, B 0.000, C 0.000 }
gfCNCPoint2[5495] = {X 369.1843, Y 20.7635, Z -2.1667, A 0.000, B 0.000, C 0.000 }
gfCNCPoint2[5496] = {X 369.4374, Y 23.4005, Z -2.1667, A 0.000, B 0.000, C 0.000 }
gfCNCPoint2[5497] = {X 369.4666, Y 26.0494, Z -2.1667, A 0.000, B 0.000, C 0.000 }
gfCNCPoint2[5498] = {X 369.2718, Y 28.6914, Z -2.1667, A 0.000, B 0.000, C 0.000 }
gfCNCPoint2[5499] = {X 368.8544, Y 31.3074, Z -2.1667, A 0.000, B 0.000, C 0.000 }
gfCNCPoint2[5500] = {X 368.3374, Y 33.3847, Z -2.1667, A 0.000, B 0.000, C 0.000 }
gfCNCPoint2[5501] = {X 367.6387, Y 35.4081, Z -2.1667, A 0.000, B 0.000, C 0.000 }
gfCNCPoint2[5502] = {X 366.7640, Y 37.3619, Z -2.1667, A 0.000, B 0.000, C 0.000 }
gfCNCPoint2[5503] = {X 365.7200, Y 39.2307, Z -2.1667, A 0.000, B 0.000, C 0.000 }
gfCNCPoint2[5504] = {X 364.5149, Y 40.9999, Z -2.1667, A 0.000, B 0.000, C 0.000 }
gfCNCPoint2[5505] = {X 363.3060, Y 42.4898, Z -2.1667, A 0.000, B 0.000, C 0.000 }
gfCNCPoint2[5506] = {X 361.9710, Y 43.8680, Z -2.1667, A 0.000, B 0.000, C 0.000 }
gfCNCPoint2[5507] = {X 360.5204, Y 45.1238, Z -2.1667, A 0.000, B 0.000, C 0.000 }
gfCNCPoint2[5508] = {X 358.9652, Y 46.2476, Z -2.1667, A 0.000, B 0.000, C 0.000 }
gfCNCPoint2[5509] = {X 357.3175, Y 47.2307, Z -2.1667, A 0.000, B 0.000, C 0.000 }
gfCNCPoint2[5510] = {X 355.3843, Y 48.1083, Z -2.1667, A 0.000, B 0.000, C 0.000 }
gfCNCPoint2[5511] = {X 353.3764, Y 48.7982, Z -2.1667, A 0.000, B 0.000, C 0.000 }
gfCNCPoint2[5512] = {X 351.3120, Y 49.2941, Z -2.1667, A 0.000, B 0.000, C 0.000 }
gfCNCPoint2[5513] = {X 349.2098, Y 49.5916, Z -2.1667, A 0.000, B 0.000, C 0.000 }
gfCNCPoint2[5514] = {X 347.0889, Y 49.6879, Z -2.1667, A 0.000, B 0.000, C 0.000 }
gfCNCPoint2[5515] = {X 345.0499, Y 49.6539, Z -2.1667, A 0.000, B 0.000, C 0.000 }
gfCNCPoint2[5516] = {X 343.0216, Y 49.4432, Z -2.1667, A 0.000, B 0.000, C 0.000 }
gfCNCPoint2[5517] = {X 341.0191, Y 49.0573, Z -2.1667, A 0.000, B 0.000, C 0.000 }
gfCNCPoint2[5518] = {X 339.0577, Y 48.4991, Z -2.1667, A 0.000, B 0.000, C 0.000 }
gfCNCPoint2[5519] = {X 337.1521, Y 47.7729, Z -2.1667, A 0.000, B 0.000, C 0.000 }
gfCNCPoint2[5520] = {X 335.3167, Y 46.8842, Z -2.1667, A 0.000, B 0.000, C 0.000 }
gfCNCPoint2[5521] = {X 333.7145, Y 45.8912, Z -2.1667, A 0.000, B 0.000, C 0.000 }
gfCNCPoint2[5522] = {X 332.1961, Y 44.7744, Z -2.1667, A 0.000, B 0.000, C 0.000 }
gfCNCPoint2[5523] = {X 330.7711, Y 43.5406, Z -2.1667, A 0.000, B 0.000, C 0.000 }
gfCNCPoint2[5524] = {X 329.8559, Y 43.5681, Z -2.1667, A 0.000, B 0.000, C 0.000 }
gfCNCPoint2[5525] = {X 328.9583, Y 43.3867, Z -2.1667, A 0.000, B 0.000, C 0.000 }
gfCNCPoint2[5526] = {X 328.1256, Y 43.0059, Z -2.1667, A 0.000, B 0.000, C 0.000 }
gfCNCPoint2[5527] = {X 327.4012, Y 42.4458, Z -2.1667, A 0.000, B 0.000, C 0.000 }
gfCNCPoint2[5528] = {X 326.8042, Y 41.8634, Z -2.1667, A 0.000, B 0.000, C 0.000 }
gfCNCPoint2[5529] = {X 326.2223, Y 41.1472, Z -2.1667, A 0.000, B 0.000, C 0.000 }
gfCNCPoint2[5530] = {X 325.8201, Y 40.3166, Z -2.1667, A 0.000, B 0.000, C 0.000 }
gfCNCPoint2[5531] = {X 325.6189, Y 39.4160, Z -2.1667, A 0.000, B 0.000, C 0.000 }
gfCNCPoint2[5532] = {X 325.6294, Y 38.4932, Z -2.1667, A 0.000, B 0.000, C 0.000 }
gfCNCPoint2[5533] = {X 325.8511, Y 37.5974, Z -2.1667, A 0.000, B 0.000, C 0.000 }
gfCNCPoint2[5534] = {X 326.2722, Y 36.7763, Z -2.1667, A 0.000, B 0.000, C 0.000 }
gfCNCPoint2[5535] = {X 330.5290, Y 30.4119, Z -2.1667, A 0.000, B 0.000, C 0.000 }
gfCNCPoint2[5536] = {X 331.0932, Y 29.7535, Z -2.1667, A 0.000, B 0.000, C 0.000 }
gfCNCPoint2[5537] = {X 331.7861, Y 29.2322, Z -2.1667, A 0.000, B 0.000, C 0.000 }
gfCNCPoint2[5538] = {X 332.5750, Y 28.8724, Z -2.1667, A 0.000, B 0.000, C 0.000 }
gfCNCPoint2[5539] = {X 333.4230, Y 28.6911, Z -2.1667, A 0.000, B 0.000, C 0.000 }
gfCNCPoint2[5540] = {X 334.2900, Y 28.6968, Z -2.1667, A 0.000, B 0.000, C 0.000 }
gfCNCPoint2[5541] = {X 335.1355, Y 28.8892, Z -2.1667, A 0.000, B 0.000, C 0.000 }
gfCNCPoint2[5542] = {X 335.9197, Y 29.2593, Z -2.1667, A 0.000, B 0.000, C 0.000 }
gfCNCPoint2[5543] = {X 336.6057, Y 29.7897, Z -2.1667, A 0.000, B 0.000, C 0.000 }
gfCNCPoint2[5544] = {X 337.2041, Y 30.3665, Z -2.1667, A 0.000, B 0.000, C 0.000 }
gfCNCPoint2[5545] = {X 337.7083, Y 30.9703, Z -2.1667, A 0.000, B 0.000, C 0.000 }
gfCNCPoint2[5546] = {X 338.0846, Y 31.6611, Z -2.1667, A 0.000, B 0.000, C 0.000 }
gfCNCPoint2[5547] = {X 338.3184, Y 32.4122, Z -2.1667, A 0.000, B 0.000, C 0.000 }
gfCNCPoint2[5548] = {X 338.4007, Y 33.1945, Z -2.1667, A 0.000, B 0.000, C 0.000 }
gfCNCPoint2[5549] = {X 338.3283, Y 33.9779, Z -2.1667, A 0.000, B 0.000, C 0.000 }
gfCNCPoint2[5550] = {X 339.1623, Y 34.7432, Z -2.1667, A 0.000, B 0.000, C 0.000 }
gfCNCPoint2[5551] = {X 340.0372, Y 35.4613, Z -2.1667, A 0.000, B 0.000, C 0.000 }
gfCNCPoint2[5552] = {X 341.2952, Y 36.2948, Z -2.1667, A 0.000, B 0.000, C 0.000 }
gfCNCPoint2[5553] = {X 342.6560, Y 36.9471, Z -2.1667, A 0.000, B 0.000, C 0.000 }
gfCNCPoint2[5554] = {X 344.0936, Y 37.4059, Z -2.1667, A 0.000, B 0.000, C 0.000 }
gfCNCPoint2[5555] = {X 345.5807, Y 37.6624, Z -2.1667, A 0.000, B 0.000, C 0.000 }
gfCNCPoint2[5556] = {X 347.0889, Y 37.7118, Z -2.1667, A 0.000, B 0.000, C 0.000 }
gfCNCPoint2[5557] = {X 347.5341, Y 37.6887, Z -2.1667, A 0.000, B 0.000, C 0.000 }
gfCNCPoint2[5558] = {X 348.7332, Y 37.5475, Z -2.1667, A 0.000, B 0.000, C 0.000 }
gfCNCPoint2[5559] = {X 349.9035, Y 37.2507, Z -2.1667, A 0.000, B 0.000, C 0.000 }
gfCNCPoint2[5560] = {X 351.0250, Y 36.8036, Z -2.1667, A 0.000, B 0.000, C 0.000 }
gfCNCPoint2[5561] = {X 352.0783, Y 36.2136, Z -2.1667, A 0.000, B 0.000, C 0.000 }
gfCNCPoint2[5562] = {X 353.0456, Y 35.4910, Z -2.1667, A 0.000, B 0.000, C 0.000 }
gfCNCPoint2[5563] = {X 354.2263, Y 34.3414, Z -2.1667, A 0.000, B 0.000, C 0.000 }
gfCNCPoint2[5564] = {X 355.2482, Y 33.0485, Z -2.1667, A 0.000, B 0.000, C 0.000 }
gfCNCPoint2[5565] = {X 356.0941, Y 31.6342, Z -2.1667, A 0.000, B 0.000, C 0.000 }
gfCNCPoint2[5566] = {X 356.7497, Y 30.1223, Z -2.1667, A 0.000, B 0.000, C 0.000 }
gfCNCPoint2[5567] = {X 357.2040, Y 28.5381, Z -2.1667, A 0.000, B 0.000, C 0.000 }
gfCNCPoint2[5568] = {X 357.4823, Y 26.8196, Z -2.1667, A 0.000, B 0.000, C 0.000 }
gfCNCPoint2[5569] = {X 357.5957, Y 25.0823, Z -2.1667, A 0.000, B 0.000, C 0.000 }
gfCNCPoint2[5570] = {X 357.5431, Y 23.3422, Z -2.1667, A 0.000, B 0.000, C 0.000 }
gfCNCPoint2[5571] = {X 357.3251, Y 21.6150, Z -2.1667, A 0.000, B 0.000, C 0.000 }
gfCNCPoint2[5572] = {X 356.9797, Y 20.1274, Z -2.1667, A 0.000, B 0.000, C 0.000 }
gfCNCPoint2[5573] = {X 356.4530, Y 18.6940, Z -2.1667, A 0.000, B 0.000, C 0.000 }
gfCNCPoint2[5574] = {X 355.7531, Y 17.3367, Z -2.1667, A 0.000, B 0.000, C 0.000 }
gfCNCPoint2[5575] = {X 354.8906, Y 16.0764, Z -2.1667, A 0.000, B 0.000, C 0.000 }
gfCNCPoint2[5576] = {X 353.9739, Y 15.0543, Z -2.1667, A 0.000, B 0.000, C 0.000 }
gfCNCPoint2[5577] = {X 352.9203, Y 14.1740, Z -2.1667, A 0.000, B 0.000, C 0.000 }
gfCNCPoint2[5578] = {X 351.7515, Y 13.4536, Z -2.1667, A 0.000, B 0.000, C 0.000 }
gfCNCPoint2[5579] = {X 350.4915, Y 12.9082, Z -2.1667, A 0.000, B 0.000, C 0.000 }
gfCNCPoint2[5580] = {X 349.1664, Y 12.5489, Z -2.1667, A 0.000, B 0.000, C 0.000 }
gfCNCPoint2[5581] = {X 347.3712, Y 12.3251, Z -2.1667, A 0.000, B 0.000, C 0.000 }
gfCNCPoint2[5582] = {X 345.5623, Y 12.3398, Z -2.1667, A 0.000, B 0.000, C 0.000 }
gfCNCPoint2[5583] = {X 343.7710, Y 12.5927, Z -2.1667, A 0.000, B 0.000, C 0.000 }
gfCNCPoint2[5584] = {X 342.0287, Y 13.0792, Z -2.1667, A 0.000, B 0.000, C 0.000 }
gfCNCPoint2[5585] = {X 340.3656, Y 13.7911, Z -2.1667, A 0.000, B 0.000, C 0.000 }
gfCNCPoint2[5586] = {X 338.8108, Y 14.7158, Z -2.1667, A 0.000, B 0.000, C 0.000 }
gfCNCPoint2[5587] = {X 338.7174, Y 14.7806, Z -2.1667, A 0.000, B 0.000, C 0.000 }
gfCNCPoint2[5588] = {X 338.6245, Y 14.8463, Z -2.1667, A 0.000, B 0.000, C 0.000 }
gfCNCPoint2[5589] = {X 338.6379, Y 15.0622, Z -2.1667, A 0.000, B 0.000, C 0.000 }
gfCNCPoint2[5590] = {X 338.5598, Y 16.0349, Z -2.1667, A 0.000, B 0.000, C 0.000 }
gfCNCPoint2[5591] = {X 338.2485, Y 16.9597, Z -2.1667, A 0.000, B 0.000, C 0.000 }
gfCNCPoint2[5592] = {X 337.7225, Y 17.7816, Z -2.1667, A 0.000, B 0.000, C 0.000 }
gfCNCPoint2[5593] = {X 337.0132, Y 18.4518, Z -2.1667, A 0.000, B 0.000, C 0.000 }
gfCNCPoint2[5594] = {X 336.3278, Y 18.9560, Z -2.1667, A 0.000, B 0.000, C 0.000 }
gfCNCPoint2[5595] = {X 335.5713, Y 19.3817, Z -2.1667, A 0.000, B 0.000, C 0.000 }
gfCNCPoint2[5596] = {X 334.7407, Y 19.6341, Z -2.1667, A 0.000, B 0.000, C 0.000 }
gfCNCPoint2[5597] = {X 333.8753, Y 19.7014, Z -2.1667, A 0.000, B 0.000, C 0.000 }
gfCNCPoint2[5598] = {X 333.0157, Y 19.5804, Z -2.1667, A 0.000, B 0.000, C 0.000 }
gfCNCPoint2[5599] = {X 332.2025, Y 19.2768, Z -2.1667, A 0.000, B 0.000, C 0.000 }
gfCNCPoint2[5600] = {X 331.4739, Y 18.8049, Z -2.1667, A 0.000, B 0.000, C 0.000 }
gfCNCPoint2[5601] = {X 330.8643, Y 18.1870, Z -2.1667, A 0.000, B 0.000, C 0.000 }
gfCNCPoint2[5602] = {X 330.4023, Y 17.4521, Z -2.1667, A 0.000, B 0.000, C 0.000 }
gfCNCPoint2[5603] = {X 326.8820, Y 10.2103, Z -2.1667, A 0.000, B 0.000, C 0.000 }
gfCNCPoint2[5604] = {X 326.5719, Y 9.3163, Z -2.1667, A 0.000, B 0.000, C 0.000 }
gfCNCPoint2[5605] = {X 326.4804, Y 8.3746, Z -2.1667, A 0.000, B 0.000, C 0.000 }
gfCNCPoint2[5606] = {X 326.6127, Y 7.4376, Z -2.1667, A 0.000, B 0.000, C 0.000 }
gfCNCPoint2[5607] = {X 326.9614, Y 6.5580, Z -2.1667, A 0.000, B 0.000, C 0.000 }
gfCNCPoint2[5608] = {X 327.5070, Y 5.7849, Z -2.1667, A 0.000, B 0.000, C 0.000 }
gfCNCPoint2[5609] = {X 328.2189, Y 5.1616, Z -2.1667, A 0.000, B 0.000, C 0.000 }
gfCNCPoint2[5610] = {X 328.8880, Y 4.7034, Z -2.1667, A 0.000, B 0.000, C 0.000 }
gfCNCPoint2[5611] = {X 329.7043, Y 4.2813, Z -2.1667, A 0.000, B 0.000, C 0.000 }
gfCNCPoint2[5612] = {X 330.5954, Y 4.0567, Z -2.1667, A 0.000, B 0.000, C 0.000 }
gfCNCPoint2[5613] = {X 331.5142, Y 4.0413, Z -2.1667, A 0.000, B 0.000, C 0.000 }
gfCNCPoint2[5614] = {X 332.4122, Y 4.2361, Z -2.1667, A 0.000, B 0.000, C 0.000 }
gfCNCPoint2[5615] = {X 332.5467, Y 4.2831, Z -2.1667, A 0.000, B 0.000, C 0.000 }
gfCNCPoint2[5616] = {X 332.6262, Y 4.2351, Z -2.1667, A 0.000, B 0.000, C 0.000 }
gfCNCPoint2[5617] = {X 332.7059, Y 4.1875, Z -2.1667, A 0.000, B 0.000, C 0.000 }
gfCNCPoint2[5618] = {X 334.1616, Y 3.3770, Z -2.1667, A 0.000, B 0.000, C 0.000 }
gfCNCPoint2[5619] = {X 335.6629, Y 2.6544, Z -2.1667, A 0.000, B 0.000, C 0.000 }
gfCNCPoint2[5620] = {X 336.0092, Y 2.5002, Z -2.1667, A 0.000, B 0.000, C 0.000 }
gfCNCPoint2[5621] = {X 338.0805, Y 1.6922, Z -2.1667, A 0.000, B 0.000, C 0.000 }
gfCNCPoint2[5622] = {X 340.2133, Y 1.0643, Z -2.1667, A 0.000, B 0.000, C 0.000 }
gfCNCPoint2[5623] = {X 342.3920, Y 0.6212, Z -2.1667, A 0.000, B 0.000, C 0.000 }
gfCNCPoint2[5624] = {X 344.6007, Y 0.3661, Z -2.1667, A 0.000, B 0.000, C 0.000 }
gfCNCPoint2[5625] = {X 346.8231, Y 0.3010, Z -2.1667, A 0.000, B 0.000, C 0.000 }
gfCNCPoint2[5626] = {X 349.0429, Y 0.4263, Z -2.1667, A 0.000, B 0.000, C 0.000 }
gfCNCPoint2[5627] = {X 351.2438, Y 0.7410, Z -2.1667, A 0.000, B 0.000, C 0.000 }
gfCNCPoint2[5628] = {X 351.5275, Y 0.7935, Z -2.1667, A 0.000, B 0.000, C 0.000 }
gfCNCPoint2[5629] = {X 352.2697, Y -3.2184, Z -2.1667, A 0.000, B 0.000, C 0.000 }
gfCNCPoint2[5630] = {X 352.2697, Y -3.2184, Z 0.8333, A 0.000, B 0.000, C 0.000 }
gfCNCPoint2[5631] = {X 352.2697, Y -3.2184, Z 11.0000, A 0.000, B 0.000, C 0.000 }
gfCNCPoint2[5632] = {X 606.0427, Y 42.9011, Z 11.0000, A 0.000, B 0.000, C 0.000 }
gfCNCPoint2[5633] = {X 606.0427, Y 42.9011, Z 0.8333, A 0.000, B 0.000, C 0.000 }
gfCNCPoint2[5634] = {X 606.0427, Y 42.9011, Z -2.1667, A 0.000, B 0.000, C 0.000 }
gfCNCPoint2[5635] = {X 603.6965, Y 47.0769, Z -2.1667, A 0.000, B 0.000, C 0.000 }
gfCNCPoint2[5636] = {X 603.6310, Y 47.1894, Z -2.1667, A 0.000, B 0.000, C 0.000 }
gfCNCPoint2[5637] = {X 603.5621, Y 47.2998, Z -2.1667, A 0.000, B 0.000, C 0.000 }
gfCNCPoint2[5638] = {X 603.0356, Y 47.9601, Z -2.1667, A 0.000, B 0.000, C 0.000 }
gfCNCPoint2[5639] = {X 602.3888, Y 48.5030, Z -2.1667, A 0.000, B 0.000, C 0.000 }
gfCNCPoint2[5640] = {X 601.6472, Y 48.9070, Z -2.1667, A 0.000, B 0.000, C 0.000 }
gfCNCPoint2[5641] = {X 600.8403, Y 49.1559, Z -2.1667, A 0.000, B 0.000, C 0.000 }
gfCNCPoint2[5642] = {X 600.0000, Y 49.2400, Z -2.1667, A 0.000, B 0.000, C 0.000 }
gfCNCPoint2[5643] = {X 593.5565, Y 49.2400, Z -2.1667, A 0.000, B 0.000, C 0.000 }
gfCNCPoint2[5644] = {X 592.6130, Y 49.1337, Z -2.1667, A 0.000, B 0.000, C 0.000 }
gfCNCPoint2[5645] = {X 591.7169, Y 48.8201, Z -2.1667, A 0.000, B 0.000, C 0.000 }
gfCNCPoint2[5646] = {X 590.9129, Y 48.3150, Z -2.1667, A 0.000, B 0.000, C 0.000 }
gfCNCPoint2[5647] = {X 590.2416, Y 47.6436, Z -2.1667, A 0.000, B 0.000, C 0.000 }
gfCNCPoint2[5648] = {X 589.7364, Y 46.8397, Z -2.1667, A 0.000, B 0.000, C 0.000 }
gfCNCPoint2[5649] = {X 589.4228, Y 45.9435, Z -2.1667, A 0.000, B 0.000, C 0.000 }
gfCNCPoint2[5650] = {X 589.3165, Y 45.0000, Z -2.1667, A 0.000, B 0.000, C 0.000 }
gfCNCPoint2[5651] = {X 589.3165, Y 44.0647, Z -2.1667, A 0.000, B 0.000, C 0.000 }
gfCNCPoint2[5652] = {X 589.4215, Y 43.1447, Z -2.1667, A 0.000, B 0.000, C 0.000 }
gfCNCPoint2[5653] = {X 589.7216, Y 42.2688, Z -2.1667, A 0.000, B 0.000, C 0.000 }
gfCNCPoint2[5654] = {X 590.2030, Y 41.4778, Z -2.1667, A 0.000, B 0.000, C 0.000 }
gfCNCPoint2[5655] = {X 590.8431, Y 40.8087, Z -2.1667, A 0.000, B 0.000, C 0.000 }
gfCNCPoint2[5656] = {X 590.8434, Y 33.1188, Z -2.1667, A 0.000, B 0.000, C 0.000 }
gfCNCPoint2[5657] = {X 585.3714, Y 46.6218, Z -2.1667, A 0.000, B 0.000, C 0.000 }
gfCNCPoint2[5658] = {X 585.0085, Y 47.3114, Z -2.1667, A 0.000, B 0.000, C 0.000 }
gfCNCPoint2[5659] = {X 584.5255, Y 47.9228, Z -2.1667, A 0.000, B 0.000, C 0.000 }
gfCNCPoint2[5660] = {X 583.9387, Y 48.4356, Z -2.1667, A 0.000, B 0.000, C 0.000 }
gfCNCPoint2[5661] = {X 583.2680, Y 48.8323, Z -2.1667, A 0.000, B 0.000, C 0.000 }
gfCNCPoint2[5662] = {X 582.3418, Y 49.1460, Z -2.1667, A 0.000, B 0.000, C 0.000 }
gfCNCPoint2[5663] = {X 581.3682, Y 49.2391, Z -2.1667, A 0.000, B 0.000, C 0.000 }
gfCNCPoint2[5664] = {X 580.3993, Y 49.1068, Z -2.1667, A 0.000, B 0.000, C 0.000 }
gfCNCPoint2[5665] = {X 579.4864, Y 48.7559, Z -2.1667, A 0.000, B 0.000, C 0.000 }
gfCNCPoint2[5666] = {X 578.6782, Y 48.2052, Z -2.1667, A 0.000, B 0.000, C 0.000 }
gfCNCPoint2[5667] = {X 578.0177, Y 47.4840, Z -2.1667, A 0.000, B 0.000, C 0.000 }
gfCNCPoint2[5668] = {X 577.5400, Y 46.6307, Z -2.1667, A 0.000, B 0.000, C 0.000 }
gfCNCPoint2[5669] = {X 571.9379, Y 32.9321, Z -2.1667, A 0.000, B 0.000, C 0.000 }
gfCNCPoint2[5670] = {X 571.9383, Y 40.8082, Z -2.1667, A 0.000, B 0.000, C 0.000 }
gfCNCPoint2[5671] = {X 572.5763, Y 41.4684, Z -2.1667, A 0.000, B 0.000, C 0.000 }
gfCNCPoint2[5672] = {X 573.0573, Y 42.2504, Z -2.1667, A 0.000, B 0.000, C 0.000 }
gfCNCPoint2[5673] = {X 573.3587, Y 43.1176, Z -2.1667, A 0.000, B 0.000, C 0.000 }
gfCNCPoint2[5674] = {X 573.4663, Y 44.0294, Z -2.1667, A 0.000, B 0.000, C 0.000 }
gfCNCPoint2[5675] = {X 573.4664, Y 45.0000, Z -2.1667, A 0.000, B 0.000, C 0.000 }
gfCNCPoint2[5676] = {X 573.3601, Y 45.9435, Z -2.1667, A 0.000, B 0.000, C 0.000 }
gfCNCPoint2[5677] = {X 573.0465, Y 46.8397, Z -2.1667, A 0.000, B 0.000, C 0.000 }
gfCNCPoint2[5678] = {X 572.5414, Y 47.6436, Z -2.1667, A 0.000, B 0.000, C 0.000 }
gfCNCPoint2[5679] = {X 571.8700, Y 48.3150, Z -2.1667, A 0.000, B 0.000, C 0.000 }
gfCNCPoint2[5680] = {X 571.0661, Y 48.8201, Z -2.1667, A 0.000, B 0.000, C 0.000 }
gfCNCPoint2[5681] = {X 570.1699, Y 49.1337, Z -2.1667, A 0.000, B 0.000, C 0.000 }
gfCNCPoint2[5682] = {X 569.2264, Y 49.2400, Z -2.1667, A 0.000, B 0.000, C 0.000 }
gfCNCPoint2[5683] = {X 562.4443, Y 49.2400, Z -2.1667, A 0.000, B 0.000, C 0.000 }
gfCNCPoint2[5684] = {X 561.5008, Y 49.1337, Z -2.1667, A 0.000, B 0.000, C 0.000 }
gfCNCPoint2[5685] = {X 560.6046, Y 48.8201, Z -2.1667, A 0.000, B 0.000, C 0.000 }
gfCNCPoint2[5686] = {X 559.8007, Y 48.3150, Z -2.1667, A 0.000, B 0.000, C 0.000 }
gfCNCPoint2[5687] = {X 559.1293, Y 47.6436, Z -2.1667, A 0.000, B 0.000, C 0.000 }
gfCNCPoint2[5688] = {X 558.6242, Y 46.8397, Z -2.1667, A 0.000, B 0.000, C 0.000 }
gfCNCPoint2[5689] = {X 558.3106, Y 45.9435, Z -2.1667, A 0.000, B 0.000, C 0.000 }
gfCNCPoint2[5690] = {X 558.2043, Y 45.0000, Z -2.1667, A 0.000, B 0.000, C 0.000 }
gfCNCPoint2[5691] = {X 558.2043, Y 44.0649, Z -2.1667, A 0.000, B 0.000, C 0.000 }
gfCNCPoint2[5692] = {X 558.3091, Y 43.1444, Z -2.1667, A 0.000, B 0.000, C 0.000 }
gfCNCPoint2[5693] = {X 558.6095, Y 42.2682, Z -2.1667, A 0.000, B 0.000, C 0.000 }
gfCNCPoint2[5694] = {X 559.0916, Y 41.4771, Z -2.1667, A 0.000, B 0.000, C 0.000 }
gfCNCPoint2[5695] = {X 559.7327, Y 40.8084, Z -2.1667, A 0.000, B 0.000, C 0.000 }
gfCNCPoint2[5696] = {X 559.7327, Y 9.1936, Z -2.1667, A 0.000, B 0.000, C 0.000 }
gfCNCPoint2[5697] = {X 559.0944, Y 8.5332, Z -2.1667, A 0.000, B 0.000, C 0.000 }
gfCNCPoint2[5698] = {X 558.6133, Y 7.7509, Z -2.1667, A 0.000, B 0.000, C 0.000 }
gfCNCPoint2[5699] = {X 558.3119, Y 6.8833, Z -2.1667, A 0.000, B 0.000, C 0.000 }
gfCNCPoint2[5700] = {X 558.2045, Y 5.9711, Z -2.1667, A 0.000, B 0.000, C 0.000 }
gfCNCPoint2[5701] = {X 558.2043, Y 5.0000, Z -2.1667, A 0.000, B 0.000, C 0.000 }
gfCNCPoint2[5702] = {X 558.3106, Y 4.0565, Z -2.1667, A 0.000, B 0.000, C 0.000 }
gfCNCPoint2[5703] = {X 558.6242, Y 3.1603, Z -2.1667, A 0.000, B 0.000, C 0.000 }
gfCNCPoint2[5704] = {X 559.1293, Y 2.3564, Z -2.1667, A 0.000, B 0.000, C 0.000 }
gfCNCPoint2[5705] = {X 559.8007, Y 1.6850, Z -2.1667, A 0.000, B 0.000, C 0.000 }
gfCNCPoint2[5706] = {X 560.6046, Y 1.1799, Z -2.1667, A 0.000, B 0.000, C 0.000 }
gfCNCPoint2[5707] = {X 561.5008, Y 0.8663, Z -2.1667, A 0.000, B 0.000, C 0.000 }
gfCNCPoint2[5708] = {X 562.4443, Y 0.7600, Z -2.1667, A 0.000, B 0.000, C 0.000 }
gfCNCPoint2[5709] = {X 570.9376, Y 0.7600, Z -2.1667, A 0.000, B 0.000, C 0.000 }
gfCNCPoint2[5710] = {X 571.8810, Y 0.8663, Z -2.1667, A 0.000, B 0.000, C 0.000 }
gfCNCPoint2[5711] = {X 572.7772, Y 1.1799, Z -2.1667, A 0.000, B 0.000, C 0.000 }
gfCNCPoint2[5712] = {X 573.5812, Y 1.6850, Z -2.1667, A 0.000, B 0.000, C 0.000 }
gfCNCPoint2[5713] = {X 574.2525, Y 2.3564, Z -2.1667, A 0.000, B 0.000, C 0.000 }
gfCNCPoint2[5714] = {X 574.7577, Y 3.1603, Z -2.1667, A 0.000, B 0.000, C 0.000 }
gfCNCPoint2[5715] = {X 575.0712, Y 4.0565, Z -2.1667, A 0.000, B 0.000, C 0.000 }
gfCNCPoint2[5716] = {X 575.1776, Y 5.0000, Z -2.1667, A 0.000, B 0.000, C 0.000 }
gfCNCPoint2[5717] = {X 575.1776, Y 5.9342, Z -2.1667, A 0.000, B 0.000, C 0.000 }
gfCNCPoint2[5718] = {X 575.1074, Y 6.7021, Z -2.1667, A 0.000, B 0.000, C 0.000 }
gfCNCPoint2[5719] = {X 574.8994, Y 7.4446, Z -2.1667, A 0.000, B 0.000, C 0.000 }
gfCNCPoint2[5720] = {X 574.5603, Y 8.1371, Z -2.1667, A 0.000, B 0.000, C 0.000 }
gfCNCPoint2[5721] = {X 574.5194, Y 8.2150, Z -2.1667, A 0.000, B 0.000, C 0.000 }
gfCNCPoint2[5722] = {X 581.1908, Y 24.5825, Z -2.1667, A 0.000, B 0.000, C 0.000 }
gfCNCPoint2[5723] = {X 587.9350, Y 8.0883, Z -2.1667, A 0.000, B 0.000, C 0.000 }
gfCNCPoint2[5724] = {X 587.6159, Y 7.4202, Z -2.1667, A 0.000, B 0.000, C 0.000 }
gfCNCPoint2[5725] = {X 587.4180, Y 6.7068, Z -2.1667, A 0.000, B 0.000, C 0.000 }
gfCNCPoint2[5726] = {X 587.3471, Y 5.9698, Z -2.1667, A 0.000, B 0.000, C 0.000 }
gfCNCPoint2[5727] = {X 587.3470, Y 5.0000, Z -2.1667, A 0.000, B 0.000, C 0.000 }
gfCNCPoint2[5728] = {X 587.4533, Y 4.0565, Z -2.1667, A 0.000, B 0.000, C 0.000 }
gfCNCPoint2[5729] = {X 587.7668, Y 3.1603, Z -2.1667, A 0.000, B 0.000, C 0.000 }
gfCNCPoint2[5730] = {X 588.2720, Y 2.3564, Z -2.1667, A 0.000, B 0.000, C 0.000 }
gfCNCPoint2[5731] = {X 588.9434, Y 1.6850, Z -2.1667, A 0.000, B 0.000, C 0.000 }
gfCNCPoint2[5732] = {X 589.7473, Y 1.1799, Z -2.1667, A 0.000, B 0.000, C 0.000 }
gfCNCPoint2[5733] = {X 590.6435, Y 0.8663, Z -2.1667, A 0.000, B 0.000, C 0.000 }
gfCNCPoint2[5734] = {X 591.5870, Y 0.7600, Z -2.1667, A 0.000, B 0.000, C 0.000 }
gfCNCPoint2[5735] = {X 600.0000, Y 0.7600, Z -2.1667, A 0.000, B 0.000, C 0.000 }
gfCNCPoint2[5736] = {X 600.8403, Y 0.8441, Z -2.1667, A 0.000, B 0.000, C 0.000 }
gfCNCPoint2[5737] = {X 601.6472, Y 1.0930, Z -2.1667, A 0.000, B 0.000, C 0.000 }
gfCNCPoint2[5738] = {X 602.3888, Y 1.4970, Z -2.1667, A 0.000, B 0.000, C 0.000 }
gfCNCPoint2[5739] = {X 603.0356, Y 2.0399, Z -2.1667, A 0.000, B 0.000, C 0.000 }
gfCNCPoint2[5740] = {X 603.5621, Y 2.7002, Z -2.1667, A 0.000, B 0.000, C 0.000 }
gfCNCPoint2[5741] = {X 603.6310, Y 2.8106, Z -2.1667, A 0.000, B 0.000, C 0.000 }
gfCNCPoint2[5742] = {X 603.6965, Y 2.9231, Z -2.1667, A 0.000, B 0.000, C 0.000 }
gfCNCPoint2[5743] = {X 607.8234, Y 10.2681, Z -2.1667, A 0.000, B 0.000, C 0.000 }
gfCNCPoint2[5744] = {X 607.8234, Y 10.2681, Z 0.8333, A 0.000, B 0.000, C 0.000 }
gfCNCPoint2[5745] = {X 607.8234, Y 10.2681, Z 11.0000, A 0.000, B 0.000, C 0.000 }
gfCNCPoint2[5746] = {X 607.6965, Y 39.1601, Z 11.0000, A 0.000, B 0.000, C 0.000 }
gfCNCPoint2[5747] = {X 607.6965, Y 39.1601, Z 0.8333, A 0.000, B 0.000, C 0.000 }
gfCNCPoint2[5748] = {X 607.6965, Y 39.1601, Z -2.1667, A 0.000, B 0.000, C 0.000 }
gfCNCPoint2[5749] = {X 603.6965, Y 46.9083, Z -2.1667, A 0.000, B 0.000, C 0.000 }
gfCNCPoint2[5750] = {X 603.5999, Y 47.0848, Z -2.1667, A 0.000, B 0.000, C 0.000 }
gfCNCPoint2[5751] = {X 603.4949, Y 47.2564, Z -2.1667, A 0.000, B 0.000, C 0.000 }
gfCNCPoint2[5752] = {X 602.9784, Y 47.9043, Z -2.1667, A 0.000, B 0.000, C 0.000 }
gfCNCPoint2[5753] = {X 602.3437, Y 48.4369, Z -2.1667, A 0.000, B 0.000, C 0.000 }
gfCNCPoint2[5754] = {X 601.6161, Y 48.8332, Z -2.1667, A 0.000, B 0.000, C 0.000 }
gfCNCPoint2[5755] = {X 600.8244, Y 49.0775, Z -2.1667, A 0.000, B 0.000, C 0.000 }
gfCNCPoint2[5756] = {X 600.0000, Y 49.1600, Z -2.1667, A 0.000, B 0.000, C 0.000 }
gfCNCPoint2[5757] = {X 593.5565, Y 49.1600, Z -2.1667, A 0.000, B 0.000, C 0.000 }
gfCNCPoint2[5758] = {X 592.6308, Y 49.0557, Z -2.1667, A 0.000, B 0.000, C 0.000 }
gfCNCPoint2[5759] = {X 591.7516, Y 48.7480, Z -2.1667, A 0.000, B 0.000, C 0.000 }
gfCNCPoint2[5760] = {X 590.9628, Y 48.2524, Z -2.1667, A 0.000, B 0.000, C 0.000 }
gfCNCPoint2[5761] = {X 590.3041, Y 47.5937, Z -2.1667, A 0.000, B 0.000, C 0.000 }
gfCNCPoint2[5762] = {X 589.8085, Y 46.8050, Z -2.1667, A 0.000, B 0.000, C 0.000 }
gfCNCPoint2[5763] = {X 589.5008, Y 45.9257, Z -2.1667, A 0.000, B 0.000, C 0.000 }
gfCNCPoint2[5764] = {X 589.3965, Y 45.0000, Z -2.1667, A 0.000, B 0.000, C 0.000 }
gfCNCPoint2[5765] = {X 589.3965, Y 44.0652, Z -2.1667, A 0.000, B 0.000, C 0.000 }
gfCNCPoint2[5766] = {X 589.5016, Y 43.1533, Z -2.1667, A 0.000, B 0.000, C 0.000 }
gfCNCPoint2[5767] = {X 589.8020, Y 42.2860, Z -2.1667, A 0.000, B 0.000, C 0.000 }
gfCNCPoint2[5768] = {X 590.2835, Y 41.5045, Z -2.1667, A 0.000, B 0.000, C 0.000 }
gfCNCPoint2[5769] = {X 590.9231, Y 40.8461, Z -2.1667, A 0.000, B 0.000, C 0.000 }
gfCNCPoint2[5770] = {X 590.9235, Y 32.7084, Z -2.1667, A 0.000, B 0.000, C 0.000 }
gfCNCPoint2[5771] = {X 585.2975, Y 46.5912, Z -2.1667, A 0.000, B 0.000, C 0.000 }
gfCNCPoint2[5772] = {X 584.9414, Y 47.2678, Z -2.1667, A 0.000, B 0.000, C 0.000 }
gfCNCPoint2[5773] = {X 584.4675, Y 47.8677, Z -2.1667, A 0.000, B 0.000, C 0.000 }
gfCNCPoint2[5774] = {X 583.8918, Y 48.3708, Z -2.1667, A 0.000, B 0.000, C 0.000 }
gfCNCPoint2[5775] = {X 583.2338, Y 48.7600, Z -2.1667, A 0.000, B 0.000, C 0.000 }
gfCNCPoint2[5776] = {X 582.3250, Y 49.0678, Z -2.1667, A 0.000, B 0.000, C 0.000 }
gfCNCPoint2[5777] = {X 581.3699, Y 49.1592, Z -2.1667, A 0.000, B 0.000, C 0.000 }
gfCNCPoint2[5778] = {X 580.4192, Y 49.0293, Z -2.1667, A 0.000, B 0.000, C 0.000 }
gfCNCPoint2[5779] = {X 579.5236, Y 48.6850, Z -2.1667, A 0.000, B 0.000, C 0.000 }
gfCNCPoint2[5780] = {X 578.7306, Y 48.1448, Z -2.1667, A 0.000, B 0.000, C 0.000 }
gfCNCPoint2[5781] = {X 578.0826, Y 47.4372, Z -2.1667, A 0.000, B 0.000, C 0.000 }
gfCNCPoint2[5782] = {X 577.6138, Y 46.5999, Z -2.1667, A 0.000, B 0.000, C 0.000 }
gfCNCPoint2[5783] = {X 571.8579, Y 32.5251, Z -2.1667, A 0.000, B 0.000, C 0.000 }
gfCNCPoint2[5784] = {X 571.8583, Y 40.8460, Z -2.1667, A 0.000, B 0.000, C 0.000 }
gfCNCPoint2[5785] = {X 572.4959, Y 41.4954, Z -2.1667, A 0.000, B 0.000, C 0.000 }
gfCNCPoint2[5786] = {X 572.9770, Y 42.2678, Z -2.1667, A 0.000, B 0.000, C 0.000 }
gfCNCPoint2[5787] = {X 573.2786, Y 43.1265, Z -2.1667, A 0.000, B 0.000, C 0.000 }
gfCNCPoint2[5788] = {X 573.3863, Y 44.0301, Z -2.1667, A 0.000, B 0.000, C 0.000 }
gfCNCPoint2[5789] = {X 573.3864, Y 45.0000, Z -2.1667, A 0.000, B 0.000, C 0.000 }
gfCNCPoint2[5790] = {X 573.2821, Y 45.9257, Z -2.1667, A 0.000, B 0.000, C 0.000 }
gfCNCPoint2[5791] = {X 572.9745, Y 46.8050, Z -2.1667, A 0.000, B 0.000, C 0.000 }
gfCNCPoint2[5792] = {X 572.4788, Y 47.5937, Z -2.1667, A 0.000, B 0.000, C 0.000 }
gfCNCPoint2[5793] = {X 571.8201, Y 48.2524, Z -2.1667, A 0.000, B 0.000, C 0.000 }
gfCNCPoint2[5794] = {X 571.0314, Y 48.7480, Z -2.1667, A 0.000, B 0.000, C 0.000 }
gfCNCPoint2[5795] = {X 570.1521, Y 49.0557, Z -2.1667, A 0.000, B 0.000, C 0.000 }
gfCNCPoint2[5796] = {X 569.2264, Y 49.1600, Z -2.1667, A 0.000, B 0.000, C 0.000 }
gfCNCPoint2[5797] = {X 562.4443, Y 49.1600, Z -2.1667, A 0.000, B 0.000, C 0.000 }
gfCNCPoint2[5798] = {X 561.5186, Y 49.0557, Z -2.1667, A 0.000, B 0.000, C 0.000 }
gfCNCPoint2[5799] = {X 560.6393, Y 48.7480, Z -2.1667, A 0.000, B 0.000, C 0.000 }
gfCNCPoint2[5800] = {X 559.8506, Y 48.2524, Z -2.1667, A 0.000, B 0.000, C 0.000 }
gfCNCPoint2[5801] = {X 559.1919, Y 47.5937, Z -2.1667, A 0.000, B 0.000, C 0.000 }
gfCNCPoint2[5802] = {X 558.6963, Y 46.8050, Z -2.1667, A 0.000, B 0.000, C 0.000 }
gfCNCPoint2[5803] = {X 558.3886, Y 45.9257, Z -2.1667, A 0.000, B 0.000, C 0.000 }
gfCNCPoint2[5804] = {X 558.2843, Y 45.0000, Z -2.1667, A 0.000, B 0.000, C 0.000 }
gfCNCPoint2[5805] = {X 558.2843, Y 44.0652, Z -2.1667, A 0.000, B 0.000, C 0.000 }
gfCNCPoint2[5806] = {X 558.3892, Y 43.1530, Z -2.1667, A 0.000, B 0.000, C 0.000 }
gfCNCPoint2[5807] = {X 558.6899, Y 42.2853, Z -2.1667, A 0.000, B 0.000, C 0.000 }
gfCNCPoint2[5808] = {X 559.1721, Y 41.5039, Z -2.1667, A 0.000, B 0.000, C 0.000 }
gfCNCPoint2[5809] = {X 559.8127, Y 40.8460, Z -2.1667, A 0.000, B 0.000, C 0.000 }
gfCNCPoint2[5810] = {X 559.8127, Y 9.1559, Z -2.1667, A 0.000, B 0.000, C 0.000 }
gfCNCPoint2[5811] = {X 559.1748, Y 8.5063, Z -2.1667, A 0.000, B 0.000, C 0.000 }
gfCNCPoint2[5812] = {X 558.6936, Y 7.7335, Z -2.1667, A 0.000, B 0.000, C 0.000 }
gfCNCPoint2[5813] = {X 558.3920, Y 6.8745, Z -2.1667, A 0.000, B 0.000, C 0.000 }
gfCNCPoint2[5814] = {X 558.2845, Y 5.9704, Z -2.1667, A 0.000, B 0.000, C 0.000 }
gfCNCPoint2[5815] = {X 558.2843, Y 5.0000, Z -2.1667, A 0.000, B 0.000, C 0.000 }
gfCNCPoint2[5816] = {X 558.3886, Y 4.0743, Z -2.1667, A 0.000, B 0.000, C 0.000 }
gfCNCPoint2[5817] = {X 558.6963, Y 3.1950, Z -2.1667, A 0.000, B 0.000, C 0.000 }
gfCNCPoint2[5818] = {X 559.1919, Y 2.4063, Z -2.1667, A 0.000, B 0.000, C 0.000 }
gfCNCPoint2[5819] = {X 559.8506, Y 1.7476, Z -2.1667, A 0.000, B 0.000, C 0.000 }
gfCNCPoint2[5820] = {X 560.6393, Y 1.2520, Z -2.1667, A 0.000, B 0.000, C 0.000 }
gfCNCPoint2[5821] = {X 561.5186, Y 0.9443, Z -2.1667, A 0.000, B 0.000, C 0.000 }
gfCNCPoint2[5822] = {X 562.4443, Y 0.8400, Z -2.1667, A 0.000, B 0.000, C 0.000 }
gfCNCPoint2[5823] = {X 570.9376, Y 0.8400, Z -2.1667, A 0.000, B 0.000, C 0.000 }
gfCNCPoint2[5824] = {X 571.8632, Y 0.9443, Z -2.1667, A 0.000, B 0.000, C 0.000 }
gfCNCPoint2[5825] = {X 572.7425, Y 1.2520, Z -2.1667, A 0.000, B 0.000, C 0.000 }
gfCNCPoint2[5826] = {X 573.5313, Y 1.7476, Z -2.1667, A 0.000, B 0.000, C 0.000 }
gfCNCPoint2[5827] = {X 574.1900, Y 2.4063, Z -2.1667, A 0.000, B 0.000, C 0.000 }
gfCNCPoint2[5828] = {X 574.6856, Y 3.1950, Z -2.1667, A 0.000, B 0.000, C 0.000 }
gfCNCPoint2[5829] = {X 574.9933, Y 4.0743, Z -2.1667, A 0.000, B 0.000, C 0.000 }
gfCNCPoint2[5830] = {X 575.0976, Y 5.0000, Z -2.1667, A 0.000, B 0.000, C 0.000 }
gfCNCPoint2[5831] = {X 575.0976, Y 5.9342, Z -2.1667, A 0.000, B 0.000, C 0.000 }
gfCNCPoint2[5832] = {X 575.0286, Y 6.6884, Z -2.1667, A 0.000, B 0.000, C 0.000 }
gfCNCPoint2[5833] = {X 574.8240, Y 7.4176, Z -2.1667, A 0.000, B 0.000, C 0.000 }
gfCNCPoint2[5834] = {X 574.4906, Y 8.0977, Z -2.1667, A 0.000, B 0.000, C 0.000 }
gfCNCPoint2[5835] = {X 574.4312, Y 8.2107, Z -2.1667, A 0.000, B 0.000, C 0.000 }
gfCNCPoint2[5836] = {X 581.1907, Y 24.7942, Z -2.1667, A 0.000, B 0.000, C 0.000 }
gfCNCPoint2[5837] = {X 588.0241, Y 8.0816, Z -2.1667, A 0.000, B 0.000, C 0.000 }
gfCNCPoint2[5838] = {X 587.7002, Y 7.4168, Z -2.1667, A 0.000, B 0.000, C 0.000 }
gfCNCPoint2[5839] = {X 587.4990, Y 6.7052, Z -2.1667, A 0.000, B 0.000, C 0.000 }
gfCNCPoint2[5840] = {X 587.4271, Y 5.9692, Z -2.1667, A 0.000, B 0.000, C 0.000 }
gfCNCPoint2[5841] = {X 587.4270, Y 5.0000, Z -2.1667, A 0.000, B 0.000, C 0.000 }
gfCNCPoint2[5842] = {X 587.5313, Y 4.0743, Z -2.1667, A 0.000, B 0.000, C 0.000 }
gfCNCPoint2[5843] = {X 587.8389, Y 3.1950, Z -2.1667, A 0.000, B 0.000, C 0.000 }
gfCNCPoint2[5844] = {X 588.3345, Y 2.4063, Z -2.1667, A 0.000, B 0.000, C 0.000 }
gfCNCPoint2[5845] = {X 588.9932, Y 1.7476, Z -2.1667, A 0.000, B 0.000, C 0.000 }
gfCNCPoint2[5846] = {X 589.7820, Y 1.2520, Z -2.1667, A 0.000, B 0.000, C 0.000 }
gfCNCPoint2[5847] = {X 590.6613, Y 0.9443, Z -2.1667, A 0.000, B 0.000, C 0.000 }
gfCNCPoint2[5848] = {X 591.5870, Y 0.8400, Z -2.1667, A 0.000, B 0.000, C 0.000 }
gfCNCPoint2[5849] = {X 600.0000, Y 0.8400, Z -2.1667, A 0.000, B 0.000, C 0.000 }
gfCNCPoint2[5850] = {X 600.8244, Y 0.9225, Z -2.1667, A 0.000, B 0.000, C 0.000 }
gfCNCPoint2[5851] = {X 601.6161, Y 1.1668, Z -2.1667, A 0.000, B 0.000, C 0.000 }
gfCNCPoint2[5852] = {X 602.3437, Y 1.5631, Z -2.1667, A 0.000, B 0.000, C 0.000 }
gfCNCPoint2[5853] = {X 602.9784, Y 2.0957, Z -2.1667, A 0.000, B 0.000, C 0.000 }
gfCNCPoint2[5854] = {X 603.4949, Y 2.7436, Z -2.1667, A 0.000, B 0.000, C 0.000 }
gfCNCPoint2[5855] = {X 603.5999, Y 2.9152, Z -2.1667, A 0.000, B 0.000, C 0.000 }
gfCNCPoint2[5856] = {X 603.6965, Y 3.0917, Z -2.1667, A 0.000, B 0.000, C 0.000 }
gfCNCPoint2[5857] = {X 607.6965, Y 10.8399, Z -2.1667, A 0.000, B 0.000, C 0.000 }
gfCNCPoint2[5858] = {X 607.6965, Y 10.8399, Z 0.8333, A 0.000, B 0.000, C 0.000 }
gfCNCPoint2[5859] = {X 607.6965, Y 10.8399, Z 11.0000, A 0.000, B 0.000, C 0.000 }
gfCNCPoint2[5860] = {X 607.6965, Y 38.1651, Z 11.0000, A 0.000, B 0.000, C 0.000 }
gfCNCPoint2[5861] = {X 607.6965, Y 38.1651, Z 0.8333, A 0.000, B 0.000, C 0.000 }
gfCNCPoint2[5862] = {X 607.6965, Y 38.1651, Z -2.1667, A 0.000, B 0.000, C 0.000 }
gfCNCPoint2[5863] = {X 603.6965, Y 46.7270, Z -2.1667, A 0.000, B 0.000, C 0.000 }
gfCNCPoint2[5864] = {X 603.5703, Y 46.9746, Z -2.1667, A 0.000, B 0.000, C 0.000 }
gfCNCPoint2[5865] = {X 603.4276, Y 47.2131, Z -2.1667, A 0.000, B 0.000, C 0.000 }
gfCNCPoint2[5866] = {X 602.9211, Y 47.8484, Z -2.1667, A 0.000, B 0.000, C 0.000 }
gfCNCPoint2[5867] = {X 602.2987, Y 48.3708, Z -2.1667, A 0.000, B 0.000, C 0.000 }
gfCNCPoint2[5868] = {X 601.5850, Y 48.7595, Z -2.1667, A 0.000, B 0.000, C 0.000 }
gfCNCPoint2[5869] = {X 600.8086, Y 48.9991, Z -2.1667, A 0.000, B 0.000, C 0.000 }
gfCNCPoint2[5870] = {X 600.0000, Y 49.0800, Z -2.1667, A 0.000, B 0.000, C 0.000 }
gfCNCPoint2[5871] = {X 593.5565, Y 49.0800, Z -2.1667, A 0.000, B 0.000, C 0.000 }
gfCNCPoint2[5872] = {X 592.6486, Y 48.9777, Z -2.1667, A 0.000, B 0.000, C 0.000 }
gfCNCPoint2[5873] = {X 591.7863, Y 48.6760, Z -2.1667, A 0.000, B 0.000, C 0.000 }
gfCNCPoint2[5874] = {X 591.0127, Y 48.1899, Z -2.1667, A 0.000, B 0.000, C 0.000 }
gfCNCPoint2[5875] = {X 590.3667, Y 47.5438, Z -2.1667, A 0.000, B 0.000, C 0.000 }
gfCNCPoint2[5876] = {X 589.8806, Y 46.7702, Z -2.1667, A 0.000, B 0.000, C 0.000 }
gfCNCPoint2[5877] = {X 589.5788, Y 45.9079, Z -2.1667, A 0.000, B 0.000, C 0.000 }
gfCNCPoint2[5878] = {X 589.4765, Y 45.0000, Z -2.1667, A 0.000, B 0.000, C 0.000 }
gfCNCPoint2[5879] = {X 589.4765, Y 44.0656, Z -2.1667, A 0.000, B 0.000, C 0.000 }
gfCNCPoint2[5880] = {X 589.5738, Y 43.1968, Z -2.1667, A 0.000, B 0.000, C 0.000 }
gfCNCPoint2[5881] = {X 589.8520, Y 42.3680, Z -2.1667, A 0.000, B 0.000, C 0.000 }
gfCNCPoint2[5882] = {X 590.2986, Y 41.6165, Z -2.1667, A 0.000, B 0.000, C 0.000 }
gfCNCPoint2[5883] = {X 590.8936, Y 40.9760, Z -2.1667, A 0.000, B 0.000, C 0.000 }
gfCNCPoint2[5884] = {X 590.9480, Y 40.9295, Z -2.1667, A 0.000, B 0.000, C 0.000 }
gfCNCPoint2[5885] = {X 591.0031, Y 40.8840, Z -2.1667, A 0.000, B 0.000, C 0.000 }
gfCNCPoint2[5886] = {X 591.0035, Y 32.2979, Z -2.1667, A 0.000, B 0.000, C 0.000 }
gfCNCPoint2[5887] = {X 585.2236, Y 46.5606, Z -2.1667, A 0.000, B 0.000, C 0.000 }
gfCNCPoint2[5888] = {X 584.8743, Y 47.2242, Z -2.1667, A 0.000, B 0.000, C 0.000 }
gfCNCPoint2[5889] = {X 584.4095, Y 47.8125, Z -2.1667, A 0.000, B 0.000, C 0.000 }
gfCNCPoint2[5890] = {X 583.8449, Y 48.3059, Z -2.1667, A 0.000, B 0.000, C 0.000 }
gfCNCPoint2[5891] = {X 583.1996, Y 48.6877, Z -2.1667, A 0.000, B 0.000, C 0.000 }
gfCNCPoint2[5892] = {X 582.3082, Y 48.9895, Z -2.1667, A 0.000, B 0.000, C 0.000 }
gfCNCPoint2[5893] = {X 581.3715, Y 49.0792, Z -2.1667, A 0.000, B 0.000, C 0.000 }
gfCNCPoint2[5894] = {X 580.4391, Y 48.9518, Z -2.1667, A 0.000, B 0.000, C 0.000 }
gfCNCPoint2[5895] = {X 579.5607, Y 48.6142, Z -2.1667, A 0.000, B 0.000, C 0.000 }
gfCNCPoint2[5896] = {X 578.7830, Y 48.0843, Z -2.1667, A 0.000, B 0.000, C 0.000 }
gfCNCPoint2[5897] = {X 578.1474, Y 47.3903, Z -2.1667, A 0.000, B 0.000, C 0.000 }
gfCNCPoint2[5898] = {X 577.6877, Y 46.5692, Z -2.1667, A 0.000, B 0.000, C 0.000 }
gfCNCPoint2[5899] = {X 571.7779, Y 32.1181, Z -2.1667, A 0.000, B 0.000, C 0.000 }
gfCNCPoint2[5900] = {X 571.7783, Y 40.8843, Z -2.1667, A 0.000, B 0.000, C 0.000 }
gfCNCPoint2[5901] = {X 571.8683, Y 40.9568, Z -2.1667, A 0.000, B 0.000, C 0.000 }
gfCNCPoint2[5902] = {X 572.4695, Y 41.5902, Z -2.1667, A 0.000, B 0.000, C 0.000 }
gfCNCPoint2[5903] = {X 572.9221, Y 42.3372, Z -2.1667, A 0.000, B 0.000, C 0.000 }
gfCNCPoint2[5904] = {X 573.2053, Y 43.1633, Z -2.1667, A 0.000, B 0.000, C 0.000 }
gfCNCPoint2[5905] = {X 573.3063, Y 44.0308, Z -2.1667, A 0.000, B 0.000, C 0.000 }
gfCNCPoint2[5906] = {X 573.3064, Y 45.0000, Z -2.1667, A 0.000, B 0.000, C 0.000 }
gfCNCPoint2[5907] = {X 573.2041, Y 45.9079, Z -2.1667, A 0.000, B 0.000, C 0.000 }
gfCNCPoint2[5908] = {X 572.9024, Y 46.7702, Z -2.1667, A 0.000, B 0.000, C 0.000 }
gfCNCPoint2[5909] = {X 572.4163, Y 47.5438, Z -2.1667, A 0.000, B 0.000, C 0.000 }
gfCNCPoint2[5910] = {X 571.7703, Y 48.1899, Z -2.1667, A 0.000, B 0.000, C 0.000 }
gfCNCPoint2[5911] = {X 570.9967, Y 48.6760, Z -2.1667, A 0.000, B 0.000, C 0.000 }
gfCNCPoint2[5912] = {X 570.1343, Y 48.9777, Z -2.1667, A 0.000, B 0.000, C 0.000 }
gfCNCPoint2[5913] = {X 569.2264, Y 49.0800, Z -2.1667, A 0.000, B 0.000, C 0.000 }
gfCNCPoint2[5914] = {X 562.4443, Y 49.0800, Z -2.1667, A 0.000, B 0.000, C 0.000 }
gfCNCPoint2[5915] = {X 561.5364, Y 48.9777, Z -2.1667, A 0.000, B 0.000, C 0.000 }
gfCNCPoint2[5916] = {X 560.6741, Y 48.6760, Z -2.1667, A 0.000, B 0.000, C 0.000 }
gfCNCPoint2[5917] = {X 559.9005, Y 48.1899, Z -2.1667, A 0.000, B 0.000, C 0.000 }
gfCNCPoint2[5918] = {X 559.2544, Y 47.5438, Z -2.1667, A 0.000, B 0.000, C 0.000 }
gfCNCPoint2[5919] = {X 558.7683, Y 46.7702, Z -2.1667, A 0.000, B 0.000, C 0.000 }
gfCNCPoint2[5920] = {X 558.4666, Y 45.9079, Z -2.1667, A 0.000, B 0.000, C 0.000 }
gfCNCPoint2[5921] = {X 558.3643, Y 45.0000, Z -2.1667, A 0.000, B 0.000, C 0.000 }
gfCNCPoint2[5922] = {X 558.3643, Y 44.0656, Z -2.1667, A 0.000, B 0.000, C 0.000 }
gfCNCPoint2[5923] = {X 558.4613, Y 43.1967, Z -2.1667, A 0.000, B 0.000, C 0.000 }
gfCNCPoint2[5924] = {X 558.7397, Y 42.3678, Z -2.1667, A 0.000, B 0.000, C 0.000 }
gfCNCPoint2[5925] = {X 559.1868, Y 41.6164, Z -2.1667, A 0.000, B 0.000, C 0.000 }
gfCNCPoint2[5926] = {X 559.7825, Y 40.9763, Z -2.1667, A 0.000, B 0.000, C 0.000 }
gfCNCPoint2[5927] = {X 559.8372, Y 40.9296, Z -2.1667, A 0.000, B 0.000, C 0.000 }
gfCNCPoint2[5928] = {X 559.8927, Y 40.8839, Z -2.1667, A 0.000, B 0.000, C 0.000 }
gfCNCPoint2[5929] = {X 559.8927, Y 9.1177, Z -2.1667, A 0.000, B 0.000, C 0.000 }
gfCNCPoint2[5930] = {X 559.8367, Y 9.0720, Z -2.1667, A 0.000, B 0.000, C 0.000 }
gfCNCPoint2[5931] = {X 559.7815, Y 9.0253, Z -2.1667, A 0.000, B 0.000, C 0.000 }
gfCNCPoint2[5932] = {X 559.1888, Y 8.3934, Z -2.1667, A 0.000, B 0.000, C 0.000 }
gfCNCPoint2[5933] = {X 558.7430, Y 7.6506, Z -2.1667, A 0.000, B 0.000, C 0.000 }
gfCNCPoint2[5934] = {X 558.4640, Y 6.8304, Z -2.1667, A 0.000, B 0.000, C 0.000 }
gfCNCPoint2[5935] = {X 558.3645, Y 5.9697, Z -2.1667, A 0.000, B 0.000, C 0.000 }
gfCNCPoint2[5936] = {X 558.3643, Y 5.0000, Z -2.1667, A 0.000, B 0.000, C 0.000 }
gfCNCPoint2[5937] = {X 558.4666, Y 4.0921, Z -2.1667, A 0.000, B 0.000, C 0.000 }
gfCNCPoint2[5938] = {X 558.7683, Y 3.2298, Z -2.1667, A 0.000, B 0.000, C 0.000 }
gfCNCPoint2[5939] = {X 559.2544, Y 2.4562, Z -2.1667, A 0.000, B 0.000, C 0.000 }
gfCNCPoint2[5940] = {X 559.9005, Y 1.8101, Z -2.1667, A 0.000, B 0.000, C 0.000 }
gfCNCPoint2[5941] = {X 560.6741, Y 1.3240, Z -2.1667, A 0.000, B 0.000, C 0.000 }
gfCNCPoint2[5942] = {X 561.5364, Y 1.0223, Z -2.1667, A 0.000, B 0.000, C 0.000 }
gfCNCPoint2[5943] = {X 562.4443, Y 0.9200, Z -2.1667, A 0.000, B 0.000, C 0.000 }
gfCNCPoint2[5944] = {X 570.9376, Y 0.9200, Z -2.1667, A 0.000, B 0.000, C 0.000 }
gfCNCPoint2[5945] = {X 571.8454, Y 1.0223, Z -2.1667, A 0.000, B 0.000, C 0.000 }
gfCNCPoint2[5946] = {X 572.7078, Y 1.3240, Z -2.1667, A 0.000, B 0.000, C 0.000 }
gfCNCPoint2[5947] = {X 573.4814, Y 1.8101, Z -2.1667, A 0.000, B 0.000, C 0.000 }
gfCNCPoint2[5948] = {X 574.1274, Y 2.4562, Z -2.1667, A 0.000, B 0.000, C 0.000 }
gfCNCPoint2[5949] = {X 574.6135, Y 3.2298, Z -2.1667, A 0.000, B 0.000, C 0.000 }
gfCNCPoint2[5950] = {X 574.9153, Y 4.0921, Z -2.1667, A 0.000, B 0.000, C 0.000 }
gfCNCPoint2[5951] = {X 575.0176, Y 5.0000, Z -2.1667, A 0.000, B 0.000, C 0.000 }
gfCNCPoint2[5952] = {X 575.0176, Y 5.9342, Z -2.1667, A 0.000, B 0.000, C 0.000 }
gfCNCPoint2[5953] = {X 574.9499, Y 6.6739, Z -2.1667, A 0.000, B 0.000, C 0.000 }
gfCNCPoint2[5954] = {X 574.7493, Y 7.3891, Z -2.1667, A 0.000, B 0.000, C 0.000 }
gfCNCPoint2[5955] = {X 574.4223, Y 8.0561, Z -2.1667, A 0.000, B 0.000, C 0.000 }
gfCNCPoint2[5956] = {X 574.3780, Y 8.1272, Z -2.1667, A 0.000, B 0.000, C 0.000 }
gfCNCPoint2[5957] = {X 574.3323, Y 8.1973, Z -2.1667, A 0.000, B 0.000, C 0.000 }
gfCNCPoint2[5958] = {X 574.3572, Y 8.2410, Z -2.1667, A 0.000, B 0.000, C 0.000 }
gfCNCPoint2[5959] = {X 581.1906, Y 25.0058, Z -2.1667, A 0.000, B 0.000, C 0.000 }
gfCNCPoint2[5960] = {X 588.1135, Y 8.0745, Z -2.1667, A 0.000, B 0.000, C 0.000 }
gfCNCPoint2[5961] = {X 587.7845, Y 7.4132, Z -2.1667, A 0.000, B 0.000, C 0.000 }
gfCNCPoint2[5962] = {X 587.5802, Y 6.7035, Z -2.1667, A 0.000, B 0.000, C 0.000 }
gfCNCPoint2[5963] = {X 587.5071, Y 5.9685, Z -2.1667, A 0.000, B 0.000, C 0.000 }
gfCNCPoint2[5964] = {X 587.5070, Y 5.0000, Z -2.1667, A 0.000, B 0.000, C 0.000 }
gfCNCPoint2[5965] = {X 587.6092, Y 4.0921, Z -2.1667, A 0.000, B 0.000, C 0.000 }
gfCNCPoint2[5966] = {X 587.9110, Y 3.2298, Z -2.1667, A 0.000, B 0.000, C 0.000 }
gfCNCPoint2[5967] = {X 588.3971, Y 2.4562, Z -2.1667, A 0.000, B 0.000, C 0.000 }
gfCNCPoint2[5968] = {X 589.0431, Y 1.8101, Z -2.1667, A 0.000, B 0.000, C 0.000 }
gfCNCPoint2[5969] = {X 589.8167, Y 1.3240, Z -2.1667, A 0.000, B 0.000, C 0.000 }
gfCNCPoint2[5970] = {X 590.6791, Y 1.0223, Z -2.1667, A 0.000, B 0.000, C 0.000 }
gfCNCPoint2[5971] = {X 591.5870, Y 0.9200, Z -2.1667, A 0.000, B 0.000, C 0.000 }
gfCNCPoint2[5972] = {X 600.0000, Y 0.9200, Z -2.1667, A 0.000, B 0.000, C 0.000 }
gfCNCPoint2[5973] = {X 600.8086, Y 1.0009, Z -2.1667, A 0.000, B 0.000, C 0.000 }
gfCNCPoint2[5974] = {X 601.5850, Y 1.2405, Z -2.1667, A 0.000, B 0.000, C 0.000 }
gfCNCPoint2[5975] = {X 602.2987, Y 1.6292, Z -2.1667, A 0.000, B 0.000, C 0.000 }
gfCNCPoint2[5976] = {X 602.9211, Y 2.1516, Z -2.1667, A 0.000, B 0.000, C 0.000 }
gfCNCPoint2[5977] = {X 603.4276, Y 2.7869, Z -2.1667, A 0.000, B 0.000, C 0.000 }
gfCNCPoint2[5978] = {X 603.5703, Y 3.0254, Z -2.1667, A 0.000, B 0.000, C 0.000 }
gfCNCPoint2[5979] = {X 603.6965, Y 3.2730, Z -2.1667, A 0.000, B 0.000, C 0.000 }
gfCNCPoint2[5980] = {X 607.6965, Y 11.8349, Z -2.1667, A 0.000, B 0.000, C 0.000 }
gfCNCPoint2[5981] = {X 607.6965, Y 11.8349, Z 0.8333, A 0.000, B 0.000, C 0.000 }
gfCNCPoint2[5982] = {X 607.6965, Y 11.8349, Z 11.0000, A 0.000, B 0.000, C 0.000 }
gfCNCPoint2[5983] = {X 607.6965, Y 36.8543, Z 11.0000, A 0.000, B 0.000, C 0.000 }
gfCNCPoint2[5984] = {X 607.6965, Y 36.8543, Z 0.8333, A 0.000, B 0.000, C 0.000 }
gfCNCPoint2[5985] = {X 607.6965, Y 36.8543, Z -2.1667, A 0.000, B 0.000, C 0.000 }
gfCNCPoint2[5986] = {X 603.6965, Y 46.5284, Z -2.1667, A 0.000, B 0.000, C 0.000 }
gfCNCPoint2[5987] = {X 603.5430, Y 46.8566, Z -2.1667, A 0.000, B 0.000, C 0.000 }
gfCNCPoint2[5988] = {X 603.3604, Y 47.1697, Z -2.1667, A 0.000, B 0.000, C 0.000 }
gfCNCPoint2[5989] = {X 602.8638, Y 47.7926, Z -2.1667, A 0.000, B 0.000, C 0.000 }
gfCNCPoint2[5990] = {X 602.2536, Y 48.3047, Z -2.1667, A 0.000, B 0.000, C 0.000 }
gfCNCPoint2[5991] = {X 601.5540, Y 48.6858, Z -2.1667, A 0.000, B 0.000, C 0.000 }
gfCNCPoint2[5992] = {X 600.7927, Y 48.9207, Z -2.1667, A 0.000, B 0.000, C 0.000 }
gfCNCPoint2[5993] = {X 600.0000, Y 49.0000, Z -2.1667, A 0.000, B 0.000, C 0.000 }
gfCNCPoint2[5994] = {X 593.5565, Y 49.0000, Z -2.1667, A 0.000, B 0.000, C 0.000 }
gfCNCPoint2[5995] = {X 592.6664, Y 48.8997, Z -2.1667, A 0.000, B 0.000, C 0.000 }
gfCNCPoint2[5996] = {X 591.8210, Y 48.6039, Z -2.1667, A 0.000, B 0.000, C 0.000 }
gfCNCPoint2[5997] = {X 591.0626, Y 48.1273, Z -2.1667, A 0.000, B 0.000, C 0.000 }
gfCNCPoint2[5998] = {X 590.4292, Y 47.4940, Z -2.1667, A 0.000, B 0.000, C 0.000 }
gfCNCPoint2[5999] = {X 589.9527, Y 46.7355, Z -2.1667, A 0.000, B 0.000, C 0.000 }
gfCNCPoint2[6000] = {X 589.6568, Y 45.8901, Z -2.1667, A 0.000, B 0.000, C 0.000 }
gfCNCPoint2[6001] = {X 589.5565, Y 45.0000, Z -2.1667, A 0.000, B 0.000, C 0.000 }
gfCNCPoint2[6002] = {X 589.5565, Y 44.0660, Z -2.1667, A 0.000, B 0.000, C 0.000 }
gfCNCPoint2[6003] = {X 589.6519, Y 43.2141, Z -2.1667, A 0.000, B 0.000, C 0.000 }
gfCNCPoint2[6004] = {X 589.9247, Y 42.4014, Z -2.1667, A 0.000, B 0.000, C 0.000 }
gfCNCPoint2[6005] = {X 590.3627, Y 41.6644, Z -2.1667, A 0.000, B 0.000, C 0.000 }
gfCNCPoint2[6006] = {X 590.9462, Y 41.0363, Z -2.1667, A 0.000, B 0.000, C 0.000 }
gfCNCPoint2[6007] = {X 591.0139, Y 40.9787, Z -2.1667, A 0.000, B 0.000, C 0.000 }
gfCNCPoint2[6008] = {X 591.0830, Y 40.9225, Z -2.1667, A 0.000, B 0.000, C 0.000 }
gfCNCPoint2[6009] = {X 591.0851, Y 40.3075, Z -2.1667, A 0.000, B 0.000, C 0.000 }
gfCNCPoint2[6010] = {X 591.0834, Y 32.0426, Z -2.1667, A 0.000, B 0.000, C 0.000 }
gfCNCPoint2[6011] = {X 590.9675, Y 32.1736, Z -2.1667, A 0.000, B 0.000, C 0.000 }
gfCNCPoint2[6012] = {X 590.3131, Y 33.7886, Z -2.1667, A 0.000, B 0.000, C 0.000 }
gfCNCPoint2[6013] = {X 585.1497, Y 46.5300, Z -2.1667, A 0.000, B 0.000, C 0.000 }
gfCNCPoint2[6014] = {X 584.8073, Y 47.1805, Z -2.1667, A 0.000, B 0.000, C 0.000 }
gfCNCPoint2[6015] = {X 584.3516, Y 47.7574, Z -2.1667, A 0.000, B 0.000, C 0.000 }
gfCNCPoint2[6016] = {X 583.7980, Y 48.2411, Z -2.1667, A 0.000, B 0.000, C 0.000 }
gfCNCPoint2[6017] = {X 583.1653, Y 48.6154, Z -2.1667, A 0.000, B 0.000, C 0.000 }
gfCNCPoint2[6018] = {X 582.2878, Y 48.9121, Z -2.1667, A 0.000, B 0.000, C 0.000 }
gfCNCPoint2[6019] = {X 581.3656, Y 48.9990, Z -2.1667, A 0.000, B 0.000, C 0.000 }
gfCNCPoint2[6020] = {X 580.4480, Y 48.8715, Z -2.1667, A 0.000, B 0.000, C 0.000 }
gfCNCPoint2[6021] = {X 579.5845, Y 48.5363, Z -2.1667, A 0.000, B 0.000, C 0.000 }
gfCNCPoint2[6022] = {X 578.8212, Y 48.0115, Z -2.1667, A 0.000, B 0.000, C 0.000 }
gfCNCPoint2[6023] = {X 578.1990, Y 47.3251, Z -2.1667, A 0.000, B 0.000, C 0.000 }
gfCNCPoint2[6024] = {X 577.7515, Y 46.5141, Z -2.1667, A 0.000, B 0.000, C 0.000 }
gfCNCPoint2[6025] = {X 571.6978, Y 31.7111, Z -2.1667, A 0.000, B 0.000, C 0.000 }
gfCNCPoint2[6026] = {X 571.6983, Y 40.9225, Z -2.1667, A 0.000, B 0.000, C 0.000 }
gfCNCPoint2[6027] = {X 571.8372, Y 41.0355, Z -2.1667, A 0.000, B 0.000, C 0.000 }
gfCNCPoint2[6028] = {X 572.4235, Y 41.6620, Z -2.1667, A 0.000, B 0.000, C 0.000 }
gfCNCPoint2[6029] = {X 572.8626, Y 42.3991, Z -2.1667, A 0.000, B 0.000, C 0.000 }
gfCNCPoint2[6030] = {X 573.1344, Y 43.2129, Z -2.1667, A 0.000, B 0.000, C 0.000 }
gfCNCPoint2[6031] = {X 573.2264, Y 44.0660, Z -2.1667, A 0.000, B 0.000, C 0.000 }
gfCNCPoint2[6032] = {X 573.2264, Y 45.0000, Z -2.1667, A 0.000, B 0.000, C 0.000 }
gfCNCPoint2[6033] = {X 573.1261, Y 45.8901, Z -2.1667, A 0.000, B 0.000, C 0.000 }
gfCNCPoint2[6034] = {X 572.8303, Y 46.7355, Z -2.1667, A 0.000, B 0.000, C 0.000 }
gfCNCPoint2[6035] = {X 572.3538, Y 47.4940, Z -2.1667, A 0.000, B 0.000, C 0.000 }
gfCNCPoint2[6036] = {X 571.7204, Y 48.1273, Z -2.1667, A 0.000, B 0.000, C 0.000 }
gfCNCPoint2[6037] = {X 570.9620, Y 48.6039, Z -2.1667, A 0.000, B 0.000, C 0.000 }
gfCNCPoint2[6038] = {X 570.1165, Y 48.8997, Z -2.1667, A 0.000, B 0.000, C 0.000 }
gfCNCPoint2[6039] = {X 569.2264, Y 49.0000, Z -2.1667, A 0.000, B 0.000, C 0.000 }
gfCNCPoint2[6040] = {X 562.4443, Y 49.0000, Z -2.1667, A 0.000, B 0.000, C 0.000 }
gfCNCPoint2[6041] = {X 561.5542, Y 48.8997, Z -2.1667, A 0.000, B 0.000, C 0.000 }
gfCNCPoint2[6042] = {X 560.7088, Y 48.6039, Z -2.1667, A 0.000, B 0.000, C 0.000 }
